C09098=1084.373,-43.335,-55.194,174.208,18.576,153.076
C09099=1084.367,-43.584,-55.182,174.206,18.574,153.076
C09100=1084.361,-43.833,-55.170,174.205,18.572,153.076
C09101=1084.355,-44.083,-55.158,174.204,18.571,153.076
C09102=1084.349,-44.333,-55.147,174.202,18.569,153.076
C09103=1084.343,-44.583,-55.134,174.201,18.568,153.076
C09104=1084.337,-44.833,-55.122,174.200,18.566,153.076
C09105=1084.331,-45.081,-55.110,174.198,18.565,153.076
C09106=1084.325,-45.331,-55.097,174.196,18.563,153.076
C09107=1084.320,-45.582,-55.086,174.195,18.561,153.076
C09108=1084.314,-45.831,-55.074,174.193,18.559,153.076
C09109=1084.308,-46.081,-55.061,174.192,18.557,153.076
C09110=1084.301,-46.330,-55.049,174.190,18.556,153.076
C09111=1084.296,-46.580,-55.038,174.189,18.554,153.076
C09112=1084.290,-46.830,-55.025,174.188,18.553,153.076
C09113=1084.284,-47.079,-55.014,174.186,18.551,153.076
C09114=1084.278,-47.329,-55.001,174.185,18.549,153.075
C09115=1084.272,-47.579,-54.990,174.183,18.547,153.075
C09116=1084.267,-47.828,-54.978,174.181,18.546,153.075
C09117=1084.260,-48.078,-54.966,174.180,18.544,153.075
C09118=1084.255,-48.327,-54.954,174.178,18.543,153.075
C09119=1084.249,-48.577,-54.942,174.177,18.541,153.075
C09120=1084.242,-48.850,-54.929,174.176,18.539,153.075
C09121=1084.236,-49.122,-54.916,174.174,18.537,153.075
C09122=1084.230,-49.395,-54.903,174.172,18.535,153.075
C09123=1084.223,-49.668,-54.890,174.171,18.534,153.075
C09124=1084.217,-49.917,-54.878,174.169,18.532,153.075
C09125=1084.211,-50.167,-54.866,174.168,18.531,153.075
C09126=1084.205,-50.416,-54.855,174.167,18.529,153.075
C09127=1084.199,-50.666,-54.842,174.164,18.527,153.075
C09128=1084.194,-50.915,-54.831,174.163,18.525,153.075
C09129=1084.187,-51.165,-54.819,174.162,18.524,153.075
C09130=1084.181,-51.415,-54.807,174.160,18.522,153.075
C09131=1084.175,-51.664,-54.796,174.158,18.521,153.075
C09132=1084.169,-51.914,-54.784,174.157,18.519,153.075
C09133=1084.163,-52.164,-54.771,174.156,18.518,153.075
C09134=1084.157,-52.413,-54.761,174.154,18.516,153.075
C09135=1084.150,-52.663,-54.749,174.153,18.515,153.075
C09136=1084.145,-52.913,-54.737,174.151,18.513,153.075
C09137=1084.139,-53.162,-54.725,174.150,18.512,153.075
C09138=1084.132,-53.412,-54.714,174.148,18.510,153.075
C09139=1084.127,-53.662,-54.702,174.147,18.509,153.075
C09140=1084.120,-53.911,-54.690,174.145,18.507,153.075
C09141=1084.114,-54.161,-54.679,174.143,18.505,153.075
C09142=1084.108,-54.410,-54.667,174.142,18.503,153.074
C09143=1084.102,-54.661,-54.655,174.140,18.502,153.074
C09144=1084.096,-54.910,-54.644,174.139,18.500,153.074
C09145=1084.090,-55.160,-54.632,174.138,18.499,153.074
C09146=1084.085,-55.409,-54.620,174.136,18.497,153.074
C09147=1084.078,-55.659,-54.609,174.135,18.496,153.074
C09148=1084.072,-55.909,-54.597,174.133,18.494,153.074
C09149=1084.066,-56.158,-54.586,174.132,18.493,153.074
C09150=1084.060,-56.408,-54.573,174.131,18.491,153.074
C09151=1084.054,-56.658,-54.563,174.129,18.490,153.074
C09152=1084.048,-56.907,-54.551,174.128,18.488,153.074
C09153=1084.042,-57.157,-54.540,174.126,18.486,153.074
C09154=1084.036,-57.407,-54.527,174.124,18.484,153.074
C09155=1084.030,-57.656,-54.516,174.123,18.483,153.074
C09156=1084.024,-57.906,-54.504,174.121,18.482,153.074
C09157=1084.018,-58.155,-54.493,174.119,18.480,153.074
C09158=1084.012,-58.405,-54.481,174.118,18.479,153.074
C09159=1084.006,-58.655,-54.470,174.117,18.477,153.074
C09160=1084.000,-58.905,-54.459,174.115,18.476,153.074
C09161=1083.993,-59.154,-54.447,174.114,18.474,153.074
C09162=1083.988,-59.404,-54.436,174.112,18.473,153.074
C09163=1083.982,-59.654,-54.423,174.111,18.471,153.074
C09164=1083.976,-59.903,-54.413,174.109,18.469,153.074
C09165=1083.970,-60.153,-54.401,174.108,18.468,153.074
C09166=1083.964,-60.402,-54.390,174.107,18.466,153.074
C09167=1083.958,-60.653,-54.378,174.105,18.465,153.074
C09168=1083.952,-60.902,-54.366,174.104,18.463,153.074
C09169=1083.946,-61.151,-54.355,174.102,18.462,153.074
C09170=1083.940,-61.401,-54.344,174.101,18.461,153.074
C09171=1083.934,-61.650,-54.333,174.099,18.459,153.074
C09172=1083.928,-61.901,-54.321,174.098,18.458,153.074
C09173=1083.922,-62.150,-54.310,174.096,18.456,153.074
C09174=1083.916,-62.400,-54.298,174.094,18.454,153.074
C09175=1083.910,-62.649,-54.287,174.093,18.452,153.074
C09176=1083.904,-62.899,-54.276,174.091,18.451,153.074
C09177=1083.899,-63.149,-54.264,174.090,18.449,153.074
C09178=1083.892,-63.399,-54.252,174.088,18.448,153.074
C09179=1083.886,-63.648,-54.241,174.087,18.447,153.074
C09180=1083.881,-63.898,-54.231,174.085,18.445,153.074
C09181=1083.874,-64.147,-54.219,174.084,18.444,153.074
C09182=1083.868,-64.397,-54.208,174.083,18.442,153.074
C09183=1083.863,-64.647,-54.196,174.081,18.441,153.074
C09184=1083.856,-64.921,-54.184,174.080,18.439,153.074
C09185=1083.850,-65.194,-54.171,174.078,18.438,153.074
C09186=1083.843,-65.469,-54.159,174.076,18.435,153.074
C09187=1083.837,-65.742,-54.147,174.075,18.434,153.073
C09188=1083.830,-65.993,-54.135,174.073,18.432,153.073
C09189=1083.824,-66.241,-54.124,174.071,18.431,153.074
C09190=1083.819,-66.491,-54.113,174.070,18.430,153.074
C09191=1083.812,-66.741,-54.102,174.069,18.428,153.073
C09192=1083.807,-66.991,-54.091,174.067,18.427,153.073
C09193=1083.800,-67.241,-54.080,174.066,18.425,153.073
C09194=1083.795,-67.490,-54.067,174.064,18.424,153.073
C09195=1083.789,-67.740,-54.056,174.063,18.422,153.073
C09196=1083.783,-67.990,-54.045,174.061,18.421,153.073
C09197=1083.777,-68.239,-54.034,174.060,18.420,153.073
C09198=1083.771,-68.489,-54.023,174.058,18.418,153.073
C09199=1083.765,-68.739,-54.012,174.057,18.416,153.073
C09200=1083.759,-68.988,-54.001,174.056,18.415,153.073
C09201=1083.753,-69.237,-53.990,174.054,18.413,153.073
C09202=1083.748,-69.488,-53.978,174.052,18.412,153.073
C09203=1083.742,-69.737,-53.967,174.051,18.411,153.073
C09204=1083.736,-69.987,-53.956,174.050,18.409,153.073
C09205=1083.730,-70.237,-53.945,174.048,18.408,153.073
C09206=1083.724,-70.486,-53.934,174.047,18.406,153.073
C09207=1083.718,-70.736,-53.923,174.045,18.405,153.073
C09208=1083.712,-70.986,-53.912,174.044,18.404,153.073
C09209=1083.706,-71.235,-53.900,174.042,18.402,153.073
C09210=1083.700,-71.484,-53.889,174.041,18.400,153.073
C09211=1083.694,-71.735,-53.878,174.039,18.399,153.073
C09212=1083.688,-71.984,-53.867,174.038,18.397,153.073
C09213=1083.683,-72.234,-53.856,174.036,18.396,153.073
C09214=1083.677,-72.483,-53.845,174.035,18.395,153.073
C09215=1083.671,-72.734,-53.834,174.033,18.393,153.073
C09216=1083.665,-72.983,-53.823,174.032,18.392,153.073
C09217=1083.660,-73.233,-53.812,174.031,18.390,153.073
C09218=1083.653,-73.483,-53.801,174.029,18.389,153.073
C09219=1083.647,-73.732,-53.790,174.028,18.388,153.073
C09220=1083.642,-73.982,-53.779,174.026,18.386,153.073
C09221=1083.636,-74.231,-53.768,174.025,18.384,153.073
C09222=1083.630,-74.481,-53.757,174.023,18.383,153.073
C09223=1083.624,-74.731,-53.746,174.022,18.382,153.073
C09224=1083.618,-74.980,-53.735,174.020,18.380,153.073
C09225=1083.611,-75.230,-53.724,174.018,18.379,153.073
C09226=1083.605,-75.480,-53.714,174.017,18.378,153.073
C09227=1083.600,-75.729,-53.703,174.016,18.376,153.073
C09228=1083.593,-75.979,-53.691,174.014,18.375,153.073
C09229=1083.588,-76.229,-53.681,174.013,18.374,153.073
C09230=1083.582,-76.478,-53.670,174.011,18.372,153.073
C09231=1083.575,-76.729,-53.658,174.009,18.371,153.073
C09232=1083.569,-76.978,-53.648,174.008,18.370,153.073
C09233=1083.563,-77.227,-53.637,174.007,18.368,153.073
C09234=1083.557,-77.477,-53.626,174.005,18.367,153.073
C09235=1083.551,-77.728,-53.616,174.003,18.365,153.073
C09236=1083.546,-77.977,-53.605,174.002,18.364,153.074
C09237=1083.540,-78.227,-53.594,174.000,18.363,153.074
C09238=1083.534,-78.476,-53.583,173.999,18.361,153.074
C09239=1083.527,-78.726,-53.573,173.997,18.360,153.074
C09240=1083.521,-78.975,-53.562,173.996,18.359,153.074
C09241=1083.516,-79.225,-53.551,173.994,18.357,153.074
C09242=1083.510,-79.474,-53.540,173.993,18.356,153.074
C09243=1083.504,-79.725,-53.529,173.991,18.355,153.074
C09244=1083.498,-79.975,-53.519,173.990,18.354,153.074
C09245=1083.492,-80.224,-53.508,173.988,18.352,153.074
C09246=1083.485,-80.474,-53.497,173.987,18.350,153.074
C09247=1083.480,-80.724,-53.486,173.985,18.349,153.074
C09248=1083.473,-81.000,-53.475,173.984,18.348,153.074
C09249=1083.466,-81.276,-53.463,173.982,18.347,153.074
C09250=1083.459,-81.552,-53.451,173.981,18.345,153.074
C09251=1083.452,-81.827,-53.440,173.979,18.344,153.074
C09252=1083.446,-82.078,-53.428,173.978,18.343,153.074
C09253=1083.440,-82.327,-53.418,173.976,18.342,153.074
C09254=1083.434,-82.577,-53.408,173.974,18.340,153.074
C09255=1083.428,-82.826,-53.397,173.973,18.339,153.074
C09256=1083.421,-83.076,-53.387,173.971,18.338,153.074
C09257=1083.416,-83.326,-53.376,173.970,18.337,153.074
C09258=1083.410,-83.575,-53.365,173.968,18.335,153.074
C09259=1083.404,-83.825,-53.355,173.967,18.334,153.074
C09260=1083.397,-84.075,-53.344,173.965,18.332,153.074
C09261=1083.392,-84.325,-53.333,173.963,18.331,153.074
C09262=1083.385,-84.574,-53.323,173.962,18.330,153.074
C09263=1083.380,-84.824,-53.313,173.960,18.329,153.074
C09264=1083.373,-85.074,-53.301,173.959,18.327,153.074
C09265=1083.367,-85.323,-53.291,173.957,18.326,153.075
C09266=1083.361,-85.573,-53.281,173.957,18.325,153.074
C09267=1083.355,-85.823,-53.271,173.955,18.324,153.075
C09268=1083.349,-86.073,-53.259,173.954,18.323,153.075
C09269=1083.343,-86.322,-53.249,173.952,18.322,153.075
C09270=1083.337,-86.572,-53.239,173.950,18.321,153.075
C09271=1083.331,-86.822,-53.228,173.949,18.319,153.075
C09272=1083.324,-87.071,-53.218,173.947,18.318,153.075
C09273=1083.318,-87.322,-53.207,173.946,18.316,153.075
C09274=1083.313,-87.571,-53.196,173.944,18.315,153.075
C09275=1083.306,-87.820,-53.186,173.943,18.314,153.075
C09276=1083.301,-88.070,-53.176,173.941,18.313,153.075
C09277=1083.294,-88.320,-53.166,173.939,18.312,153.075
C09278=1083.289,-88.569,-53.155,173.938,18.310,153.075
C09279=1083.282,-88.820,-53.145,173.936,18.309,153.075
C09280=1083.276,-89.069,-53.134,173.936,18.308,153.075
C09281=1083.271,-89.319,-53.124,173.934,18.307,153.075
C09282=1083.264,-89.568,-53.114,173.932,18.306,153.075
C09283=1083.258,-89.818,-53.103,173.931,18.305,153.075
C09284=1083.252,-90.068,-53.093,173.929,18.304,153.075
C09285=1083.246,-90.318,-53.082,173.928,18.302,153.075
C09286=1083.240,-90.568,-53.072,173.926,18.301,153.075
C09287=1083.234,-90.817,-53.061,173.925,18.299,153.075
C09288=1083.227,-91.066,-53.051,173.923,18.298,153.076
C09289=1083.222,-91.316,-53.041,173.921,18.297,153.076
C09290=1083.216,-91.566,-53.030,173.920,18.296,153.076
C09291=1083.210,-91.816,-53.021,173.919,18.295,153.076
C09292=1083.204,-92.065,-53.010,173.917,18.294,153.076
C09293=1083.198,-92.316,-53.000,173.916,18.293,153.076
C09294=1083.192,-92.565,-52.989,173.914,18.292,153.076
C09295=1083.186,-92.815,-52.979,173.913,18.290,153.076
C09296=1083.180,-93.064,-52.968,173.911,18.289,153.076
C09297=1083.174,-93.314,-52.959,173.909,18.288,153.076
C09298=1083.168,-93.564,-52.948,173.908,18.287,153.076
C09299=1083.162,-93.814,-52.938,173.906,18.286,153.076
C09300=1083.156,-94.063,-52.928,173.905,18.285,153.076
C09301=1083.150,-94.313,-52.918,173.904,18.284,153.076
C09302=1083.144,-94.562,-52.907,173.902,18.283,153.076
C09303=1083.138,-94.812,-52.897,173.901,18.281,153.076
C09304=1083.132,-95.062,-52.886,173.899,18.280,153.076
C09305=1083.126,-95.312,-52.877,173.898,18.279,153.077
C09306=1083.120,-95.562,-52.866,173.896,18.278,153.077
C09307=1083.114,-95.811,-52.856,173.895,18.276,153.077
C09308=1083.108,-96.061,-52.845,173.893,18.275,153.077
C09309=1083.102,-96.311,-52.836,173.891,18.274,153.077
C09310=1083.096,-96.561,-52.826,173.890,18.273,153.077
C09311=1083.090,-96.810,-52.815,173.889,18.272,153.077
C09312=1083.084,-97.089,-52.804,173.887,18.271,153.077
C09313=1083.077,-97.366,-52.793,173.885,18.270,153.077
C09314=1083.070,-97.645,-52.782,173.883,18.268,153.077
C09315=1083.063,-97.923,-52.770,173.882,18.267,153.077
C09316=1083.057,-98.173,-52.760,173.880,18.266,153.077
C09317=1083.051,-98.423,-52.749,173.878,18.265,153.077
C09318=1083.045,-98.672,-52.740,173.878,18.264,153.077
C09319=1083.039,-98.922,-52.730,173.876,18.263,153.077
C09320=1083.033,-99.172,-52.719,173.874,18.262,153.078
C09321=1083.027,-99.422,-52.710,173.873,18.261,153.078
C09322=1083.020,-99.672,-52.700,173.871,18.260,153.078
C09323=1083.014,-99.921,-52.690,173.870,18.258,153.078
C09324=1083.009,-100.171,-52.680,173.868,18.257,153.078
C09325=1083.002,-100.421,-52.670,173.867,18.257,153.078
C09326=1082.996,-100.670,-52.660,173.865,18.256,153.078
C09327=1082.990,-100.920,-52.650,173.864,18.255,153.078
C09328=1082.984,-101.170,-52.640,173.862,18.254,153.078
C09329=1082.978,-101.419,-52.630,173.860,18.253,153.078
C09330=1082.972,-101.669,-52.620,173.859,18.251,153.078
C09331=1082.966,-101.919,-52.610,173.857,18.250,153.079
C09332=1082.960,-102.168,-52.600,173.856,18.250,153.079
C09333=1082.954,-102.418,-52.590,173.855,18.249,153.079
C09334=1082.948,-102.668,-52.580,173.853,18.248,153.079
C09335=1082.942,-102.918,-52.570,173.851,18.247,153.079
C09336=1082.935,-103.167,-52.560,173.850,18.246,153.079
C09337=1082.929,-103.417,-52.551,173.848,18.244,153.079
C09338=1082.924,-103.667,-52.540,173.847,18.243,153.079
C09339=1082.918,-103.917,-52.531,173.846,18.242,153.079
C09340=1082.911,-104.166,-52.520,173.844,18.241,153.079
C09341=1082.905,-104.416,-52.511,173.842,18.240,153.079
C09342=1082.900,-104.666,-52.501,173.841,18.239,153.080
C09343=1082.893,-104.916,-52.491,173.839,18.238,153.080
C09344=1082.887,-105.165,-52.481,173.837,18.237,153.080
C09345=1082.881,-105.415,-52.471,173.837,18.237,153.080
C09346=1082.875,-105.665,-52.462,173.835,18.236,153.080
C09347=1082.869,-105.915,-52.452,173.833,18.235,153.080
C09348=1082.863,-106.165,-52.442,173.832,18.234,153.080
C09349=1082.857,-106.414,-52.432,173.830,18.232,153.080
C09350=1082.850,-106.664,-52.422,173.828,18.231,153.080
C09351=1082.844,-106.913,-52.413,173.828,18.231,153.080
C09352=1082.839,-107.164,-52.402,173.826,18.230,153.080
C09353=1082.833,-107.413,-52.393,173.824,18.229,153.081
C09354=1082.826,-107.663,-52.383,173.823,18.228,153.081
C09355=1082.820,-107.912,-52.373,173.821,18.227,153.081
C09356=1082.814,-108.162,-52.363,173.819,18.226,153.081
C09357=1082.808,-108.412,-52.354,173.818,18.225,153.081
C09358=1082.801,-108.662,-52.344,173.817,18.224,153.081
C09359=1082.795,-108.911,-52.335,173.815,18.223,153.081
C09360=1082.790,-109.162,-52.325,173.813,18.222,153.081
C09361=1082.784,-109.411,-52.315,173.812,18.221,153.081
C09362=1082.777,-109.661,-52.305,173.810,18.220,153.082
C09363=1082.771,-109.910,-52.295,173.809,18.220,153.082
C09364=1082.765,-110.160,-52.286,173.807,18.219,153.082
C09365=1082.759,-110.410,-52.276,173.806,18.218,153.082
C09366=1082.752,-110.660,-52.267,173.804,18.217,153.082
C09367=1082.746,-110.910,-52.257,173.802,18.216,153.082
C09368=1082.741,-111.159,-52.248,173.801,18.215,153.082
C09369=1082.735,-111.408,-52.238,173.800,18.214,153.082
C09370=1082.728,-111.658,-52.229,173.798,18.213,153.083
C09371=1082.722,-111.908,-52.219,173.796,18.212,153.083
C09372=1082.716,-112.158,-52.209,173.795,18.211,153.083
C09373=1082.710,-112.408,-52.200,173.794,18.211,153.083
C09374=1082.704,-112.658,-52.190,173.792,18.210,153.083
C09375=1082.698,-112.908,-52.180,173.790,18.209,153.083
C09376=1082.692,-113.181,-52.169,173.789,18.208,153.083
C09377=1082.684,-113.457,-52.159,173.787,18.207,153.083
C09378=1082.678,-113.731,-52.149,173.785,18.206,153.084
C09379=1082.671,-114.007,-52.138,173.783,18.205,153.084
C09380=1082.665,-114.256,-52.129,173.782,18.204,153.084
C09381=1082.659,-114.505,-52.119,173.781,18.203,153.084
C09382=1082.653,-114.755,-52.110,173.779,18.202,153.084
C09383=1082.647,-115.005,-52.100,173.778,18.201,153.084
C09384=1082.641,-115.255,-52.090,173.776,18.201,153.084
C09385=1082.635,-115.505,-52.081,173.774,18.200,153.084
C09386=1082.628,-115.754,-52.071,173.773,18.199,153.085
C09387=1082.622,-116.004,-52.062,173.771,18.198,153.085
C09388=1082.616,-116.254,-52.052,173.770,18.197,153.085
C09389=1082.609,-116.504,-52.043,173.768,18.196,153.085
C09390=1082.603,-116.753,-52.034,173.766,18.196,153.085
C09391=1082.597,-117.002,-52.024,173.765,18.195,153.085
C09392=1082.591,-117.252,-52.015,173.764,18.194,153.085
C09393=1082.585,-117.502,-52.005,173.762,18.193,153.085
C09394=1082.579,-117.752,-51.996,173.760,18.192,153.086
C09395=1082.573,-118.002,-51.987,173.759,18.192,153.086
C09396=1082.567,-118.252,-51.977,173.758,18.191,153.086
C09397=1082.561,-118.502,-51.968,173.756,18.190,153.086
C09398=1082.555,-118.752,-51.958,173.754,18.189,153.086
C09399=1082.549,-119.001,-51.949,173.753,18.189,153.086
C09400=1082.543,-119.251,-51.939,173.751,18.188,153.086
C09401=1082.536,-119.500,-51.930,173.750,18.187,153.087
C09402=1082.530,-119.750,-51.922,173.748,18.186,153.087
C09403=1082.524,-120.000,-51.912,173.746,18.186,153.087
C09404=1082.518,-120.250,-51.902,173.745,18.185,153.087
C09405=1082.512,-120.500,-51.893,173.744,18.184,153.087
C09406=1082.506,-120.749,-51.884,173.742,18.184,153.087
C09407=1082.500,-120.999,-51.874,173.740,18.183,153.088
C09408=1082.494,-121.248,-51.865,173.739,18.182,153.088
C09409=1082.487,-121.499,-51.856,173.737,18.181,153.088
C09410=1082.481,-121.748,-51.847,173.736,18.181,153.088
C09411=1082.475,-121.998,-51.837,173.734,18.180,153.088
C09412=1082.469,-122.247,-51.828,173.733,18.179,153.088
C09413=1082.463,-122.497,-51.818,173.731,18.179,153.088
C09414=1082.457,-122.748,-51.810,173.729,18.177,153.089
C09415=1082.450,-122.997,-51.801,173.728,18.176,153.089
C09416=1082.444,-123.247,-51.791,173.727,18.176,153.089
C09417=1082.438,-123.497,-51.781,173.725,18.175,153.089
C09418=1082.433,-123.746,-51.773,173.723,18.174,153.089
C09419=1082.426,-123.996,-51.763,173.721,18.174,153.089
C09420=1082.420,-124.246,-51.754,173.720,18.173,153.089
C09421=1082.413,-124.495,-51.745,173.719,18.172,153.090
C09422=1082.407,-124.746,-51.736,173.717,18.172,153.090
C09423=1082.402,-124.995,-51.727,173.716,18.171,153.090
C09424=1082.396,-125.245,-51.717,173.714,18.171,153.090
C09425=1082.389,-125.494,-51.708,173.712,18.170,153.090
C09426=1082.383,-125.745,-51.699,173.711,18.169,153.090
C09427=1082.377,-125.994,-51.690,173.710,18.169,153.091
C09428=1082.370,-126.243,-51.681,173.708,18.168,153.091
C09429=1082.364,-126.493,-51.672,173.706,18.167,153.091
C09430=1082.358,-126.743,-51.663,173.704,18.166,153.091
C09431=1082.352,-126.993,-51.653,173.703,18.166,153.091
C09432=1082.345,-127.243,-51.644,173.702,18.165,153.091
C09433=1082.340,-127.492,-51.636,173.700,18.164,153.092
C09434=1082.334,-127.742,-51.626,173.699,18.164,153.092
C09435=1082.327,-127.992,-51.617,173.697,18.163,153.092
C09436=1082.323,-128.248,-51.608,173.695,18.162,153.092
C09437=1082.323,-128.504,-51.596,173.695,18.160,153.092
C09438=1082.327,-128.758,-51.583,173.694,18.156,153.091
C09439=1082.334,-129.010,-51.570,173.694,18.152,153.090
C09440=1081.933,-129.032,-51.707,173.650,18.270,153.120
C09441=1081.926,-128.780,-51.721,173.650,18.275,153.121
C09442=1081.923,-128.525,-51.734,173.651,18.278,153.122
C09443=1081.922,-128.271,-51.745,173.652,18.280,153.122
C09444=1081.927,-128.014,-51.756,173.653,18.282,153.122
C09445=1081.932,-127.764,-51.764,173.655,18.283,153.122
C09446=1081.939,-127.515,-51.773,173.656,18.283,153.122
C09447=1081.945,-127.265,-51.783,173.658,18.284,153.122
C09448=1081.951,-127.015,-51.792,173.659,18.285,153.122
C09449=1081.957,-126.765,-51.801,173.661,18.285,153.121
C09450=1081.963,-126.516,-51.810,173.662,18.286,153.121
C09451=1081.969,-126.266,-51.819,173.664,18.286,153.121
C09452=1081.976,-126.016,-51.828,173.666,18.287,153.121
C09453=1081.982,-125.766,-51.837,173.667,18.287,153.121
C09454=1081.989,-125.517,-51.847,173.668,18.288,153.121
C09455=1081.994,-125.267,-51.855,173.670,18.289,153.120
C09456=1082.000,-125.017,-51.865,173.672,18.290,153.120
C09457=1082.007,-124.768,-51.874,173.673,18.290,153.120
C09458=1082.013,-124.517,-51.883,173.675,18.291,153.120
C09459=1082.019,-124.267,-51.892,173.676,18.292,153.120
C09460=1082.025,-124.018,-51.901,173.678,18.293,153.120
C09461=1082.031,-123.769,-51.910,173.679,18.293,153.120
C09462=1082.037,-123.518,-51.919,173.681,18.294,153.119
C09463=1082.044,-123.269,-51.929,173.683,18.295,153.119
C09464=1082.050,-123.019,-51.938,173.684,18.296,153.119
C09465=1082.056,-122.769,-51.948,173.685,18.296,153.119
C09466=1082.061,-122.520,-51.957,173.687,18.297,153.119
C09467=1082.068,-122.270,-51.965,173.689,18.298,153.119
C09468=1082.074,-122.020,-51.975,173.691,18.298,153.118
C09469=1082.080,-121.770,-51.984,173.692,18.299,153.118
C09470=1082.087,-121.520,-51.994,173.693,18.300,153.118
C09471=1082.093,-121.271,-52.004,173.695,18.301,153.118
C09472=1082.098,-121.021,-52.012,173.697,18.302,153.118
C09473=1082.104,-120.771,-52.022,173.698,18.302,153.118
C09474=1082.111,-120.522,-52.031,173.699,18.303,153.118
C09475=1082.117,-120.272,-52.040,173.701,18.304,153.117
C09476=1082.123,-120.022,-52.050,173.703,18.305,153.117
C09477=1082.130,-119.772,-52.059,173.705,18.306,153.117
C09478=1082.135,-119.523,-52.068,173.706,18.306,153.117
C09479=1082.141,-119.273,-52.077,173.707,18.307,153.117
C09480=1082.147,-119.023,-52.087,173.709,18.308,153.117
C09481=1082.153,-118.773,-52.096,173.711,18.309,153.117
C09482=1082.160,-118.524,-52.105,173.712,18.309,153.116
C09483=1082.166,-118.274,-52.115,173.713,18.310,153.116
C09484=1082.173,-118.024,-52.125,173.715,18.311,153.116
C09485=1082.179,-117.774,-52.134,173.717,18.312,153.116
C09486=1082.184,-117.525,-52.143,173.718,18.312,153.116
C09487=1082.191,-117.275,-52.153,173.719,18.313,153.116
C09488=1082.196,-117.025,-52.162,173.721,18.314,153.116
C09489=1082.203,-116.775,-52.171,173.723,18.315,153.116
C09490=1082.209,-116.525,-52.181,173.725,18.316,153.115
C09491=1082.215,-116.276,-52.190,173.726,18.316,153.115
C09492=1082.221,-116.026,-52.200,173.727,18.317,153.115
C09493=1082.227,-115.776,-52.210,173.729,18.318,153.115
C09494=1082.233,-115.526,-52.219,173.731,18.319,153.115
C09495=1082.239,-115.277,-52.228,173.732,18.320,153.115
C09496=1082.245,-115.027,-52.238,173.733,18.321,153.115
C09497=1082.251,-114.778,-52.248,173.735,18.321,153.114
C09498=1082.257,-114.528,-52.257,173.737,18.322,153.114
C09499=1082.264,-114.278,-52.267,173.738,18.323,153.114
C09500=1082.270,-114.028,-52.276,173.740,18.324,153.114
C09501=1082.277,-113.753,-52.287,173.742,18.325,153.114
C09502=1082.283,-113.478,-52.297,173.744,18.326,153.114
C09503=1082.290,-113.203,-52.308,173.744,18.327,153.114
C09504=1082.297,-112.928,-52.318,173.746,18.328,153.114
C09505=1082.303,-112.679,-52.327,173.748,18.329,153.114
C09506=1082.309,-112.429,-52.337,173.749,18.330,153.113
C09507=1082.315,-112.179,-52.346,173.751,18.331,153.113
C09508=1082.321,-111.929,-52.356,173.753,18.332,153.113
C09509=1082.328,-111.679,-52.366,173.754,18.333,153.113
C09510=1082.334,-111.430,-52.375,173.755,18.334,153.113
C09511=1082.340,-111.181,-52.385,173.757,18.334,153.113
C09512=1082.346,-110.930,-52.396,173.759,18.335,153.113
C09513=1082.352,-110.681,-52.405,173.761,18.336,153.113
C09514=1082.358,-110.431,-52.415,173.762,18.337,153.112
C09515=1082.364,-110.181,-52.424,173.763,18.338,153.112
C09516=1082.370,-109.931,-52.434,173.765,18.339,153.112
C09517=1082.377,-109.681,-52.443,173.766,18.340,153.112
C09518=1082.383,-109.432,-52.453,173.768,18.341,153.112
C09519=1082.389,-109.182,-52.463,173.770,18.342,153.112
C09520=1082.395,-108.932,-52.472,173.771,18.343,153.112
C09521=1082.402,-108.683,-52.482,173.772,18.343,153.112
C09522=1082.407,-108.434,-52.492,173.774,18.344,153.112
C09523=1082.413,-108.184,-52.501,173.776,18.345,153.111
C09524=1082.419,-107.934,-52.511,173.777,18.346,153.111
C09525=1082.425,-107.684,-52.521,173.779,18.347,153.111
C09526=1082.431,-107.434,-52.530,173.780,18.348,153.111
C09527=1082.437,-107.184,-52.540,173.782,18.349,153.111
C09528=1082.444,-106.935,-52.550,173.783,18.350,153.111
C09529=1082.450,-106.685,-52.560,173.785,18.351,153.111
C09530=1082.455,-106.435,-52.570,173.786,18.352,153.111
C09531=1082.461,-106.186,-52.580,173.788,18.353,153.111
C09532=1082.468,-105.936,-52.589,173.789,18.354,153.111
C09533=1082.474,-105.687,-52.599,173.791,18.355,153.111
C09534=1082.480,-105.437,-52.609,173.792,18.356,153.110
C09535=1082.486,-105.187,-52.619,173.794,18.357,153.110
C09536=1082.492,-104.937,-52.629,173.796,18.358,153.110
C09537=1082.498,-104.687,-52.638,173.797,18.359,153.110
C09538=1082.505,-104.438,-52.649,173.799,18.361,153.110
C09539=1082.510,-104.188,-52.659,173.800,18.361,153.110
C09540=1082.516,-103.938,-52.668,173.801,18.362,153.110
C09541=1082.522,-103.688,-52.678,173.803,18.363,153.110
C09542=1082.529,-103.439,-52.688,173.805,18.364,153.110
C09543=1082.534,-103.189,-52.698,173.806,18.365,153.110
C09544=1082.540,-102.939,-52.708,173.808,18.366,153.109
C09545=1082.547,-102.689,-52.717,173.809,18.368,153.110
C09546=1082.553,-102.440,-52.728,173.810,18.368,153.109
C09547=1082.559,-102.190,-52.738,173.812,18.369,153.109
C09548=1082.565,-101.940,-52.747,173.814,18.370,153.109
C09549=1082.571,-101.691,-52.758,173.815,18.371,153.109
C09550=1082.577,-101.441,-52.767,173.817,18.372,153.109
C09551=1082.583,-101.191,-52.777,173.818,18.374,153.109
C09552=1082.590,-100.941,-52.788,173.820,18.375,153.109
C09553=1082.596,-100.691,-52.798,173.821,18.375,153.109
C09554=1082.601,-100.441,-52.808,173.823,18.376,153.109
C09555=1082.608,-100.192,-52.818,173.824,18.377,153.109
C09556=1082.614,-99.942,-52.828,173.826,18.379,153.109
C09557=1082.620,-99.692,-52.838,173.827,18.380,153.109
C09558=1082.626,-99.443,-52.848,173.829,18.381,153.108
C09559=1082.632,-99.193,-52.858,173.831,18.382,153.108
C09560=1082.638,-98.944,-52.867,173.832,18.382,153.108
C09561=1082.644,-98.694,-52.878,173.833,18.384,153.108
C09562=1082.650,-98.444,-52.888,173.835,18.385,153.108
C09563=1082.656,-98.194,-52.897,173.836,18.386,153.108
C09564=1082.662,-97.945,-52.908,173.838,18.387,153.108
C09565=1082.670,-97.666,-52.919,173.839,18.389,153.108
C09566=1082.676,-97.388,-52.931,173.841,18.390,153.108
C09567=1082.683,-97.109,-52.942,173.843,18.391,153.108
C09568=1082.689,-96.830,-52.953,173.844,18.392,153.108
C09569=1082.695,-96.581,-52.964,173.846,18.393,153.108
C09570=1082.702,-96.331,-52.973,173.848,18.394,153.108
C09571=1082.707,-96.082,-52.984,173.849,18.396,153.108
C09572=1082.714,-95.832,-52.994,173.851,18.397,153.107
C09573=1082.719,-95.582,-53.004,173.852,18.398,153.107
C09574=1082.725,-95.333,-53.014,173.854,18.399,153.107
C09575=1082.731,-95.083,-53.025,173.855,18.400,153.107
C09576=1082.737,-94.833,-53.034,173.857,18.402,153.107
C09577=1082.743,-94.583,-53.045,173.858,18.402,153.107
C09578=1082.749,-94.334,-53.055,173.859,18.403,153.107
C09579=1082.755,-94.083,-53.065,173.861,18.405,153.107
C09580=1082.761,-93.834,-53.076,173.863,18.406,153.107
C09581=1082.767,-93.584,-53.086,173.864,18.407,153.107
C09582=1082.773,-93.334,-53.097,173.866,18.409,153.107
C09583=1082.779,-93.085,-53.106,173.867,18.410,153.107
C09584=1082.785,-92.835,-53.117,173.869,18.411,153.107
C09585=1082.791,-92.586,-53.127,173.870,18.412,153.107
C09586=1082.797,-92.336,-53.138,173.872,18.413,153.107
C09587=1082.803,-92.087,-53.148,173.874,18.415,153.107
C09588=1082.809,-91.837,-53.158,173.874,18.415,153.107
C09589=1082.816,-91.587,-53.169,173.876,18.417,153.107
C09590=1082.821,-91.337,-53.179,173.877,18.418,153.106
C09591=1082.828,-91.087,-53.189,173.879,18.419,153.106
C09592=1082.833,-90.837,-53.199,173.881,18.420,153.106
C09593=1082.840,-90.588,-53.210,173.882,18.421,153.106
C09594=1082.845,-90.339,-53.220,173.884,18.423,153.106
C09595=1082.851,-90.089,-53.231,173.885,18.424,153.106
C09596=1082.858,-89.839,-53.241,173.887,18.426,153.106
C09597=1082.863,-89.589,-53.251,173.888,18.427,153.106
C09598=1082.870,-89.339,-53.262,173.890,18.428,153.106
C09599=1082.875,-89.090,-53.273,173.892,18.429,153.106
C09600=1082.882,-88.840,-53.282,173.892,18.430,153.106
C09601=1082.887,-88.591,-53.293,173.894,18.431,153.106
C09602=1082.893,-88.340,-53.304,173.896,18.432,153.106
C09603=1082.900,-88.091,-53.314,173.897,18.434,153.106
C09604=1082.906,-87.841,-53.325,173.899,18.435,153.106
C09605=1082.912,-87.591,-53.334,173.900,18.436,153.106
C09606=1082.918,-87.342,-53.345,173.902,18.437,153.106
C09607=1082.923,-87.092,-53.356,173.903,18.439,153.106
C09608=1082.930,-86.842,-53.366,173.905,18.440,153.106
C09609=1082.936,-86.592,-53.377,173.906,18.441,153.106
C09610=1082.942,-86.343,-53.387,173.908,18.442,153.106
C09611=1082.948,-86.094,-53.398,173.909,18.444,153.106
C09612=1082.954,-85.843,-53.409,173.911,18.445,153.105
C09613=1082.961,-85.594,-53.419,173.912,18.447,153.106
C09614=1082.966,-85.344,-53.430,173.913,18.447,153.105
C09615=1082.972,-85.094,-53.439,173.915,18.449,153.106
C09616=1082.978,-84.845,-53.450,173.916,18.450,153.105
C09617=1082.985,-84.595,-53.461,173.918,18.451,153.105
C09618=1082.991,-84.346,-53.472,173.920,18.452,153.105
C09619=1082.996,-84.095,-53.482,173.921,18.454,153.105
C09620=1083.003,-83.846,-53.492,173.923,18.455,153.105
C09621=1083.009,-83.596,-53.503,173.924,18.456,153.105
C09622=1083.015,-83.347,-53.514,173.926,18.457,153.105
C09623=1083.021,-83.097,-53.524,173.927,18.459,153.105
C09624=1083.027,-82.847,-53.535,173.929,18.460,153.105
C09625=1083.033,-82.597,-53.546,173.930,18.461,153.105
C09626=1083.040,-82.348,-53.556,173.932,18.462,153.105
C09627=1083.045,-82.098,-53.567,173.933,18.464,153.105
C09628=1083.051,-81.848,-53.578,173.935,18.465,153.105
C09629=1083.058,-81.573,-53.590,173.937,18.467,153.105
C09630=1083.065,-81.296,-53.601,173.938,18.468,153.105
C09631=1083.072,-81.020,-53.613,173.940,18.469,153.105
C09632=1083.078,-80.743,-53.625,173.941,18.471,153.105
C09633=1083.085,-80.494,-53.635,173.943,18.472,153.105
C09634=1083.091,-80.244,-53.646,173.944,18.473,153.105
C09635=1083.097,-79.995,-53.657,173.946,18.475,153.105
C09636=1083.104,-79.745,-53.668,173.947,18.476,153.105
C09637=1083.109,-79.495,-53.678,173.949,18.477,153.105
C09638=1083.115,-79.245,-53.689,173.950,18.479,153.105
C09639=1083.121,-78.996,-53.700,173.952,18.480,153.105
C09640=1083.127,-78.745,-53.711,173.953,18.481,153.105
C09641=1083.133,-78.496,-53.722,173.955,18.483,153.105
C09642=1083.139,-78.247,-53.732,173.956,18.484,153.105
C09643=1083.145,-77.997,-53.743,173.958,18.485,153.105
C09644=1083.151,-77.747,-53.754,173.959,18.487,153.105
C09645=1083.157,-77.498,-53.765,173.961,18.488,153.105
C09646=1083.163,-77.248,-53.776,173.962,18.490,153.105
C09647=1083.169,-76.997,-53.786,173.964,18.491,153.105
C09648=1083.175,-76.748,-53.797,173.965,18.492,153.105
C09649=1083.181,-76.499,-53.808,173.967,18.494,153.105
C09650=1083.187,-76.249,-53.819,173.968,18.495,153.105
C09651=1083.193,-75.999,-53.830,173.970,18.496,153.104
C09652=1083.199,-75.749,-53.841,173.971,18.498,153.105
C09653=1083.204,-75.500,-53.852,173.973,18.499,153.105
C09654=1083.211,-75.250,-53.863,173.974,18.501,153.105
C09655=1083.217,-75.000,-53.874,173.976,18.502,153.104
C09656=1083.223,-74.751,-53.884,173.977,18.503,153.105
C09657=1083.229,-74.501,-53.895,173.979,18.505,153.105
C09658=1083.235,-74.251,-53.906,173.980,18.506,153.104
C09659=1083.241,-74.002,-53.917,173.982,18.508,153.104
C09660=1083.247,-73.752,-53.928,173.983,18.509,153.104
C09661=1083.253,-73.502,-53.939,173.985,18.511,153.105
C09662=1083.259,-73.253,-53.950,173.986,18.512,153.105
C09663=1083.264,-73.003,-53.961,173.988,18.513,153.104
C09664=1083.271,-72.753,-53.972,173.989,18.515,153.104
C09665=1083.276,-72.504,-53.983,173.991,18.516,153.105
C09666=1083.281,-72.254,-53.994,173.992,18.518,153.105
C09667=1083.288,-72.004,-54.006,173.994,18.519,153.105
C09668=1083.294,-71.755,-54.017,173.995,18.521,153.105
C09669=1083.300,-71.505,-54.028,173.997,18.522,153.105
C09670=1083.305,-71.256,-54.039,173.998,18.523,153.105
C09671=1083.312,-71.006,-54.050,174.000,18.525,153.105
C09672=1083.317,-70.756,-54.061,174.001,18.527,153.105
C09673=1083.323,-70.507,-54.072,174.002,18.528,153.105
C09674=1083.330,-70.256,-54.083,174.004,18.530,153.105
C09675=1083.335,-70.007,-54.094,174.005,18.531,153.105
C09676=1083.341,-69.757,-54.105,174.007,18.533,153.105
C09677=1083.347,-69.507,-54.117,174.008,18.534,153.105
C09678=1083.353,-69.258,-54.128,174.010,18.535,153.105
C09679=1083.358,-69.009,-54.139,174.011,18.537,153.105
C09680=1083.365,-68.758,-54.151,174.013,18.538,153.105
C09681=1083.370,-68.509,-54.161,174.014,18.540,153.105
C09682=1083.376,-68.259,-54.172,174.015,18.541,153.105
C09683=1083.383,-68.009,-54.184,174.017,18.543,153.105
C09684=1083.388,-67.760,-54.194,174.018,18.545,153.105
C09685=1083.394,-67.511,-54.207,174.020,18.546,153.105
C09686=1083.400,-67.260,-54.218,174.021,18.547,153.105
C09687=1083.406,-67.011,-54.229,174.023,18.549,153.105
C09688=1083.412,-66.761,-54.240,174.024,18.550,153.105
C09689=1083.418,-66.511,-54.251,174.026,18.552,153.105
C09690=1083.424,-66.262,-54.262,174.027,18.553,153.105
C09691=1083.430,-66.012,-54.274,174.029,18.555,153.105
C09692=1083.436,-65.763,-54.285,174.030,18.556,153.105
C09693=1083.442,-65.488,-54.298,174.032,18.558,153.105
C09694=1083.448,-65.214,-54.310,174.034,18.560,153.105
C09695=1083.455,-64.940,-54.323,174.035,18.561,153.105
C09696=1083.462,-64.666,-54.335,174.037,18.563,153.105
C09697=1083.468,-64.416,-54.346,174.038,18.565,153.105
C09698=1083.474,-64.167,-54.357,174.039,18.566,153.105
C09699=1083.480,-63.918,-54.368,174.041,18.568,153.105
C09700=1083.486,-63.668,-54.380,174.043,18.569,153.105
C09701=1083.491,-63.418,-54.391,174.045,18.571,153.105
C09702=1083.498,-63.168,-54.403,174.046,18.572,153.105
C09703=1083.503,-62.919,-54.414,174.048,18.574,153.105
C09704=1083.510,-62.669,-54.425,174.049,18.575,153.105
C09705=1083.515,-62.419,-54.436,174.051,18.577,153.105
C09706=1083.521,-62.169,-54.449,174.052,18.578,153.105
C09707=1083.527,-61.920,-54.460,174.053,18.580,153.105
C09708=1083.533,-61.670,-54.470,174.055,18.581,153.105
C09709=1083.540,-61.421,-54.482,174.056,18.583,153.105
C09710=1083.545,-61.171,-54.493,174.058,18.585,153.105
C09711=1083.551,-60.921,-54.506,174.059,18.586,153.105
C09712=1083.557,-60.672,-54.517,174.061,18.588,153.105
C09713=1083.563,-60.422,-54.528,174.062,18.589,153.105
C09714=1083.569,-60.173,-54.540,174.063,18.591,153.105
C09715=1083.576,-59.923,-54.551,174.065,18.592,153.106
C09716=1083.581,-59.673,-54.562,174.066,18.594,153.106
C09717=1083.587,-59.423,-54.574,174.068,18.595,153.106
C09718=1083.593,-59.174,-54.585,174.069,18.597,153.106
C09719=1083.600,-58.924,-54.597,174.071,18.598,153.106
C09720=1083.605,-58.674,-54.609,174.073,18.600,153.106
C09721=1083.611,-58.425,-54.620,174.074,18.601,153.106
C09722=1083.617,-58.175,-54.631,174.076,18.603,153.106
C09723=1083.623,-57.925,-54.643,174.077,18.605,153.106
C09724=1083.629,-57.676,-54.655,174.079,18.606,153.106
C09725=1083.635,-57.426,-54.666,174.080,18.608,153.106
C09726=1083.642,-57.176,-54.678,174.082,18.609,153.106
C09727=1083.647,-56.927,-54.689,174.083,18.611,153.106
C09728=1083.653,-56.677,-54.701,174.084,18.612,153.106
C09729=1083.659,-56.427,-54.712,174.086,18.614,153.106
C09730=1083.666,-56.178,-54.724,174.087,18.615,153.106
C09731=1083.671,-55.928,-54.735,174.089,18.617,153.106
C09732=1083.677,-55.678,-54.748,174.090,18.618,153.106
C09733=1083.683,-55.429,-54.759,174.092,18.620,153.106
C09734=1083.690,-55.179,-54.771,174.093,18.621,153.106
C09735=1083.696,-54.929,-54.782,174.095,18.624,153.106
C09736=1083.701,-54.680,-54.794,174.097,18.625,153.106
C09737=1083.708,-54.430,-54.805,174.098,18.627,153.106
C09738=1083.714,-54.181,-54.817,174.100,18.628,153.106
C09739=1083.720,-53.931,-54.829,174.101,18.630,153.106
C09740=1083.726,-53.681,-54.841,174.102,18.631,153.106
C09741=1083.732,-53.432,-54.852,174.104,18.633,153.106
C09742=1083.738,-53.182,-54.863,174.105,18.634,153.106
C09743=1083.744,-52.933,-54.876,174.107,18.636,153.106
C09744=1083.750,-52.682,-54.887,174.108,18.637,153.106
C09745=1083.757,-52.433,-54.899,174.109,18.639,153.106
C09746=1083.762,-52.184,-54.911,174.111,18.641,153.107
C09747=1083.768,-51.933,-54.922,174.112,18.643,153.107
C09748=1083.775,-51.684,-54.934,174.115,18.645,153.107
C09749=1083.780,-51.435,-54.946,174.116,18.646,153.107
C09750=1083.787,-51.184,-54.958,174.117,18.648,153.107
C09751=1083.793,-50.936,-54.969,174.119,18.649,153.107
C09752=1083.798,-50.685,-54.981,174.120,18.651,153.107
C09753=1083.805,-50.436,-54.993,174.122,18.652,153.107
C09754=1083.811,-50.187,-55.005,174.123,18.654,153.107
C09755=1083.817,-49.936,-55.016,174.125,18.655,153.107
C09756=1083.822,-49.687,-55.029,174.126,18.657,153.107
C09757=1083.829,-49.414,-55.042,174.128,18.659,153.107
C09758=1083.835,-49.141,-55.055,174.129,18.661,153.107
C09759=1083.842,-48.869,-55.068,174.131,18.663,153.107
C09760=1083.848,-48.596,-55.081,174.132,18.664,153.107
C09761=1083.854,-48.346,-55.093,174.134,18.667,153.107
C09762=1083.860,-48.096,-55.105,174.136,18.668,153.107
C09763=1083.866,-47.847,-55.117,174.137,18.670,153.107
C09764=1083.872,-47.598,-55.129,174.139,18.671,153.107
C09765=1083.877,-47.348,-55.140,174.140,18.673,153.107
C09766=1083.884,-47.098,-55.152,174.141,18.674,153.107
C09767=1083.890,-46.848,-55.165,174.143,18.676,153.108
C09768=1083.895,-46.599,-55.177,174.144,18.678,153.108
C09769=1083.901,-46.349,-55.188,174.146,18.679,153.108
C09770=1083.907,-46.100,-55.200,174.148,18.681,153.108
C09771=1083.913,-45.850,-55.212,174.149,18.683,153.108
C09772=1083.919,-45.600,-55.225,174.150,18.685,153.108
C09773=1083.924,-45.351,-55.236,174.152,18.687,153.108
C09774=1083.931,-45.101,-55.248,174.153,18.688,153.108
C09775=1083.937,-44.851,-55.261,174.155,18.690,153.108
C09776=1083.943,-44.602,-55.272,174.156,18.691,153.108
C09777=1083.949,-44.352,-55.285,174.157,18.693,153.108
C09778=1083.954,-44.102,-55.297,174.159,18.695,153.108
C09779=1083.960,-43.853,-55.308,174.161,18.697,153.108
C09780=1083.966,-43.603,-55.321,174.162,18.698,153.108
C09781=1083.972,-43.353,-55.333,174.164,18.700,153.108
C09782=1083.978,-43.104,-55.345,174.165,18.702,153.108
C09783=1083.984,-42.854,-55.358,174.167,18.704,153.108
C09784=1083.990,-42.605,-55.370,174.168,18.705,153.108
C09785=1083.996,-42.355,-55.381,174.169,18.707,153.109
C09786=1084.002,-42.105,-55.394,174.171,18.709,153.109
C09787=1084.008,-41.856,-55.406,174.173,18.711,153.109
C09788=1084.014,-41.606,-55.418,174.174,18.712,153.109
C09789=1084.020,-41.357,-55.430,174.176,18.714,153.109
C09790=1084.026,-41.107,-55.442,174.177,18.715,153.109
C09791=1084.032,-40.857,-55.455,174.178,18.717,153.109
C09792=1084.038,-40.608,-55.467,174.180,18.719,153.109
C09793=1084.044,-40.358,-55.479,174.181,18.720,153.109
C09794=1084.050,-40.108,-55.492,174.183,18.722,153.109
C09795=1084.056,-39.859,-55.504,174.185,18.724,153.109
C09796=1084.062,-39.610,-55.516,174.186,18.726,153.109
C09797=1084.068,-39.359,-55.528,174.188,18.728,153.109
C09798=1084.074,-39.109,-55.540,174.189,18.729,153.109
C09799=1084.080,-38.860,-55.552,174.190,18.731,153.109
C09800=1084.085,-38.611,-55.564,174.192,18.733,153.110
C09801=1084.091,-38.361,-55.577,174.193,18.734,153.110
C09802=1084.097,-38.111,-55.589,174.195,18.736,153.110
C09803=1084.103,-37.862,-55.602,174.196,18.738,153.110
C09804=1084.109,-37.612,-55.614,174.198,18.740,153.110
C09805=1084.115,-37.362,-55.626,174.199,18.741,153.110
C09806=1084.121,-37.112,-55.639,174.201,18.743,153.110
C09807=1084.126,-36.863,-55.651,174.202,18.745,153.110
C09808=1084.132,-36.613,-55.663,174.203,18.747,153.110
C09809=1084.138,-36.363,-55.676,174.205,18.749,153.110
C09810=1084.144,-36.115,-55.689,174.207,18.751,153.110
C09811=1084.150,-35.865,-55.701,174.208,18.752,153.110
C09812=1084.156,-35.615,-55.713,174.210,18.754,153.110
C09813=1084.162,-35.365,-55.726,174.211,18.756,153.111
C09814=1084.168,-35.116,-55.738,174.212,18.757,153.111
C09815=1084.173,-34.866,-55.751,174.214,18.759,153.111
C09816=1084.179,-34.616,-55.763,174.216,18.761,153.111
C09817=1084.185,-34.367,-55.776,174.217,18.763,153.111
C09818=1084.191,-34.117,-55.788,174.219,18.764,153.111
C09819=1084.197,-33.867,-55.800,174.220,18.767,153.111
C09820=1084.203,-33.618,-55.812,174.221,18.768,153.111
C09821=1084.209,-33.345,-55.827,174.223,18.771,153.111
C09822=1084.216,-33.074,-55.840,174.225,18.772,153.111
C09823=1084.222,-32.801,-55.854,174.226,18.774,153.111
C09824=1084.229,-32.529,-55.868,174.228,18.776,153.111
C09825=1084.235,-32.279,-55.880,174.230,18.778,153.111
C09826=1084.240,-32.030,-55.893,174.231,18.780,153.112
C09827=1084.246,-31.780,-55.905,174.232,18.781,153.112
C09828=1084.252,-31.530,-55.918,174.234,18.783,153.112
C09829=1084.258,-31.280,-55.931,174.235,18.785,153.112
C09830=1084.265,-31.031,-55.943,174.237,18.787,153.112
C09831=1084.271,-30.781,-55.955,174.239,18.789,153.112
C09832=1084.276,-30.532,-55.968,174.240,18.791,153.112
C09833=1084.282,-30.282,-55.980,174.241,18.792,153.112
C09834=1084.288,-30.033,-55.993,174.243,18.794,153.112
C09835=1084.294,-29.783,-56.006,174.244,18.796,153.112
C09836=1084.300,-29.533,-56.019,174.246,18.798,153.112
C09837=1084.306,-29.283,-56.031,174.248,18.799,153.112
C09838=1084.311,-29.034,-56.044,174.249,18.801,153.112
C09839=1084.317,-28.785,-56.057,174.250,18.803,153.113
C09840=1084.323,-28.535,-56.069,174.252,18.804,153.113
C09841=1084.329,-28.285,-56.082,174.253,18.806,153.113
C09842=1084.335,-28.036,-56.095,174.255,18.808,153.113
C09843=1084.341,-27.786,-56.108,174.257,18.810,153.113
C09844=1084.347,-27.536,-56.120,174.258,18.812,153.113
C09845=1084.353,-27.287,-56.133,174.259,18.814,153.113
C09846=1084.359,-27.037,-56.146,174.261,18.815,153.113
C09847=1084.365,-26.787,-56.158,174.263,18.818,153.113
C09848=1084.371,-26.538,-56.171,174.264,18.819,153.113
C09849=1084.377,-26.288,-56.184,174.265,18.821,153.113
C09850=1084.383,-26.038,-56.196,174.267,18.823,153.113
C09851=1084.389,-25.789,-56.210,174.268,18.825,153.114
C09852=1084.395,-25.539,-56.222,174.269,18.826,153.114
C09853=1084.400,-25.290,-56.234,174.272,18.828,153.114
C09854=1084.405,-25.041,-56.248,174.273,18.830,153.114
C09855=1084.411,-24.791,-56.261,174.274,18.832,153.114
C09856=1084.417,-24.541,-56.273,174.275,18.834,153.114
C09857=1084.423,-24.292,-56.287,174.277,18.836,153.114
C09858=1084.429,-24.042,-56.299,174.279,18.838,153.114
C09859=1084.436,-23.792,-56.313,174.280,18.840,153.114
C09860=1084.441,-23.542,-56.326,174.281,18.842,153.114
C09861=1084.446,-23.293,-56.338,174.283,18.843,153.114
C09862=1084.452,-23.044,-56.351,174.284,18.845,153.115
C09863=1084.458,-22.794,-56.364,174.286,18.847,153.115
C09864=1084.464,-22.545,-56.377,174.288,18.849,153.115
C09865=1084.470,-22.295,-56.390,174.289,18.851,153.115
C09866=1084.476,-22.045,-56.403,174.290,18.852,153.115
C09867=1084.482,-21.795,-56.416,174.292,18.855,153.115
C09868=1084.488,-21.545,-56.429,174.294,18.857,153.115
C09869=1084.494,-21.296,-56.442,174.295,18.858,153.115
C09870=1084.500,-21.046,-56.454,174.297,18.860,153.115
C09871=1084.505,-20.797,-56.468,174.298,18.862,153.115
C09872=1084.511,-20.547,-56.480,174.299,18.864,153.116
C09873=1084.517,-20.298,-56.494,174.301,18.865,153.116
C09874=1084.523,-20.048,-56.506,174.303,18.868,153.116
C09875=1084.529,-19.799,-56.519,174.304,18.869,153.116
C09876=1084.534,-19.549,-56.533,174.305,18.871,153.116
C09877=1084.540,-19.300,-56.546,174.307,18.873,153.116
C09878=1084.546,-19.050,-56.558,174.309,18.875,153.116
C09879=1084.552,-18.800,-56.572,174.310,18.877,153.116
C09880=1084.559,-18.551,-56.585,174.312,18.879,153.116
C09881=1084.564,-18.301,-56.598,174.313,18.881,153.116
C09882=1084.570,-18.052,-56.611,174.314,18.882,153.116
C09883=1084.576,-17.802,-56.624,174.316,18.885,153.117
C09884=1084.582,-17.553,-56.637,174.318,18.886,153.117
C09885=1084.589,-17.279,-56.652,174.319,18.888,153.117
C09886=1084.595,-17.007,-56.666,174.321,18.890,153.117
C09887=1084.602,-16.733,-56.680,174.322,18.892,153.117
C09888=1084.608,-16.460,-56.694,174.324,18.894,153.117
C09889=1084.613,-16.210,-56.708,174.326,18.896,153.117
C09890=1084.619,-15.961,-56.721,174.327,18.898,153.117
C09891=1084.625,-15.711,-56.734,174.329,18.900,153.117
C09892=1084.631,-15.461,-56.748,174.330,18.902,153.117
C09893=1084.638,-15.212,-56.761,174.331,18.904,153.118
C09894=1084.644,-14.962,-56.774,174.333,18.906,153.118
C09895=1084.649,-14.712,-56.788,174.335,18.908,153.118
C09896=1084.655,-14.462,-56.800,174.336,18.909,153.118
C09897=1084.661,-14.214,-56.813,174.337,18.911,153.118
C09898=1084.666,-13.964,-56.827,174.340,18.913,153.118
C09899=1084.672,-13.715,-56.840,174.341,18.915,153.118
C09900=1084.677,-13.465,-56.854,174.342,18.917,153.118
C09901=1084.684,-13.215,-56.867,174.343,18.919,153.118
C09902=1084.689,-12.966,-56.881,174.345,18.920,153.118
C09903=1084.695,-12.716,-56.893,174.347,18.923,153.119
C09904=1084.701,-12.467,-56.907,174.348,18.925,153.119
C09905=1084.707,-12.216,-56.921,174.349,18.927,153.119
C09906=1084.713,-11.967,-56.934,174.351,18.928,153.119
C09907=1084.719,-11.717,-56.947,174.353,18.931,153.119
C09908=1084.725,-11.468,-56.960,174.354,18.932,153.119
C09909=1084.730,-11.218,-56.974,174.356,18.934,153.119
C09910=1084.737,-10.969,-56.988,174.357,18.936,153.119
C09911=1084.742,-10.719,-57.001,174.358,18.938,153.119
C09912=1084.748,-10.469,-57.014,174.360,18.940,153.119
C09913=1084.753,-10.220,-57.028,174.362,18.942,153.120
C09914=1084.760,-9.971,-57.041,174.363,18.943,153.120
C09915=1084.765,-9.721,-57.055,174.364,18.945,153.120
C09916=1084.771,-9.471,-57.068,174.367,18.947,153.120
C09917=1084.777,-9.222,-57.081,174.368,18.950,153.120
C09918=1084.783,-8.972,-57.095,174.369,18.951,153.120
C09919=1084.789,-8.723,-57.108,174.370,18.953,153.120
C09920=1084.794,-8.473,-57.122,174.373,18.955,153.120
C09921=1084.801,-8.224,-57.135,174.374,18.957,153.120
C09922=1084.806,-7.974,-57.148,174.375,18.959,153.121
C09923=1084.813,-7.724,-57.162,174.377,18.961,153.121
C09924=1084.818,-7.474,-57.176,174.379,18.963,153.121
C09925=1084.824,-7.225,-57.189,174.380,18.965,153.121
C09926=1084.830,-6.976,-57.203,174.381,18.967,153.121
C09927=1084.836,-6.726,-57.216,174.383,18.968,153.121
C09928=1084.841,-6.477,-57.230,174.384,18.970,153.121
C09929=1084.847,-6.227,-57.244,174.386,18.972,153.121
C09930=1084.853,-5.978,-57.257,174.387,18.975,153.121
C09931=1084.859,-5.728,-57.271,174.389,18.976,153.121
C09932=1084.865,-5.478,-57.285,174.390,18.978,153.122
C09933=1084.871,-5.228,-57.298,174.392,18.980,153.122
C09934=1084.877,-4.979,-57.311,174.393,18.982,153.122
C09935=1084.882,-4.729,-57.325,174.395,18.984,153.122
C09936=1084.888,-4.480,-57.338,174.396,18.986,153.122
C09937=1084.894,-4.230,-57.352,174.398,18.988,153.122
C09938=1084.901,-3.980,-57.366,174.400,18.990,153.122
C09939=1084.906,-3.731,-57.380,174.401,18.991,153.122
C09940=1084.912,-3.482,-57.393,174.402,18.993,153.122
C09941=1084.918,-3.232,-57.407,174.405,18.995,153.122
C09942=1084.923,-2.982,-57.421,174.406,18.997,153.123
C09943=1084.929,-2.733,-57.434,174.407,18.999,153.123
C09944=1084.935,-2.484,-57.448,174.408,19.001,153.123
C09945=1084.941,-2.233,-57.462,174.411,19.003,153.123
C09946=1084.947,-1.984,-57.476,174.412,19.005,153.123
C09947=1084.952,-1.734,-57.490,174.413,19.007,153.123
C09948=1084.959,-1.486,-57.504,174.414,19.009,153.123
C09949=1084.964,-1.210,-57.519,174.417,19.011,153.123
C09950=1084.971,-0.935,-57.534,174.418,19.013,153.123
C09951=1084.977,-0.661,-57.550,174.420,19.016,153.124
C09952=1084.984,-0.386,-57.564,174.421,19.017,153.124
C09953=1084.989,-0.136,-57.578,174.423,19.020,153.124
C09954=1084.995,0.113,-57.592,174.425,19.021,153.124
C09955=1085.001,0.363,-57.605,174.426,19.023,153.124
C09956=1085.007,0.612,-57.620,174.427,19.025,153.124
C09957=1085.013,0.862,-57.634,174.429,19.028,153.124
C09958=1085.018,1.111,-57.648,174.431,19.030,153.124
C09959=1085.024,1.361,-57.662,174.432,19.031,153.124
C09960=1085.030,1.610,-57.675,174.434,19.034,153.125
C09961=1085.035,1.860,-57.689,174.435,19.036,153.125
C09962=1085.041,2.109,-57.703,174.437,19.037,153.125
C09963=1085.047,2.359,-57.718,174.438,19.039,153.125
C09964=1085.053,2.609,-57.732,174.440,19.041,153.125
C09965=1085.058,2.858,-57.746,174.441,19.043,153.125
C09966=1085.064,3.108,-57.759,174.443,19.045,153.125
C09967=1085.070,3.357,-57.773,174.444,19.047,153.125
C09968=1085.076,3.607,-57.788,174.446,19.049,153.125
C09969=1085.082,3.856,-57.802,174.448,19.051,153.126
C09970=1085.087,4.106,-57.815,174.449,19.053,153.126
C09971=1085.093,4.355,-57.829,174.451,19.055,153.126
C09972=1085.099,4.605,-57.843,174.452,19.057,153.126
C09973=1085.105,4.854,-57.858,174.454,19.059,153.126
C09974=1085.111,5.104,-57.871,174.455,19.061,153.126
C09975=1085.116,5.354,-57.885,174.457,19.063,153.126
C09976=1085.122,5.604,-57.899,174.458,19.065,153.126
C09977=1085.128,5.853,-57.914,174.460,19.067,153.126
C09978=1085.133,6.102,-57.928,174.461,19.068,153.127
C09979=1085.140,6.352,-57.941,174.463,19.071,153.127
C09980=1085.146,6.601,-57.956,174.464,19.072,153.127
C09981=1085.151,6.851,-57.970,174.466,19.074,153.127
C09982=1085.157,7.100,-57.984,174.468,19.076,153.127
C09983=1085.163,7.349,-57.998,174.469,19.078,153.127
C09984=1085.169,7.600,-58.013,174.470,19.080,153.127
C09985=1085.174,7.849,-58.027,174.472,19.082,153.127
C09986=1085.180,8.098,-58.041,174.474,19.085,153.127
C09987=1085.186,8.348,-58.055,174.475,19.086,153.127
C09988=1085.192,8.598,-58.069,174.476,19.088,153.128
C09989=1085.198,8.847,-58.083,174.479,19.090,153.128
C09990=1085.204,9.096,-58.097,174.480,19.092,153.128
C09991=1085.210,9.347,-58.111,174.481,19.094,153.128
C09992=1085.216,9.595,-58.126,174.483,19.096,153.128
C09993=1085.221,9.845,-58.140,174.485,19.098,153.128
C09994=1085.227,10.095,-58.155,174.486,19.100,153.128
C09995=1085.233,10.344,-58.169,174.488,19.101,153.128
C09996=1085.238,10.594,-58.182,174.490,19.104,153.128
//INST
///DATE 2021/06/17 10:54
///ATTR SC,RW,RJ
////FRAME ROBOT
///GROUP1 RB1
NOP
MOVL C00000 V=800.0 PL=0
MOVL C00001 V=800.0 PL=0
MOVL C00002 V=800.0 PL=0
MOVL C00003 V=800.0 PL=0
MOVL C00004 V=800.0 PL=0
MOVL C00005 V=800.0 PL=0
MOVL C00006 V=800.0 PL=0
MOVL C00007 V=800.0 PL=0
MOVL C00008 V=800.0 PL=0
MOVL C00009 V=800.0 PL=0
MOVL C00010 V=800.0 PL=0
MOVL C00011 V=800.0 PL=0
MOVL C00012 V=800.0 PL=0
MOVL C00013 V=800.0 PL=0
MOVL C00014 V=800.0 PL=0
MOVL C00015 V=800.0 PL=0
MOVL C00016 V=800.0 PL=0
MOVL C00017 V=800.0 PL=0
MOVL C00018 V=800.0 PL=0
MOVL C00019 V=800.0 PL=0
MOVL C00020 V=800.0 PL=0
MOVL C00021 V=800.0 PL=0
MOVL C00022 V=800.0 PL=0
MOVL C00023 V=800.0 PL=0
MOVL C00024 V=800.0 PL=0
MOVL C00025 V=800.0 PL=0
MOVL C00026 V=800.0 PL=0
MOVL C00027 V=800.0 PL=0
MOVL C00028 V=800.0 PL=0
MOVL C00029 V=800.0 PL=0
MOVL C00030 V=800.0 PL=0
MOVL C00031 V=800.0 PL=0
MOVL C00032 V=800.0 PL=0
MOVL C00033 V=800.0 PL=0
MOVL C00034 V=800.0 PL=0
MOVL C00035 V=800.0 PL=0
MOVL C00036 V=800.0 PL=0
MOVL C00037 V=800.0 PL=0
MOVL C00038 V=800.0 PL=0
MOVL C00039 V=800.0 PL=0
MOVL C00040 V=800.0 PL=0
MOVL C00041 V=800.0 PL=0
MOVL C00042 V=800.0 PL=0
MOVL C00043 V=800.0 PL=0
MOVL C00044 V=800.0 PL=0
MOVL C00045 V=800.0 PL=0
MOVL C00046 V=800.0 PL=0
MOVL C00047 V=800.0 PL=0
MOVL C00048 V=800.0 PL=0
MOVL C00049 V=800.0 PL=0
MOVL C00050 V=800.0 PL=0
MOVL C00051 V=800.0 PL=0
MOVL C00052 V=800.0 PL=0
MOVL C00053 V=800.0 PL=0
MOVL C00054 V=800.0 PL=0
MOVL C00055 V=800.0 PL=0
MOVL C00056 V=800.0 PL=0
MOVL C00057 V=800.0 PL=0
MOVL C00058 V=800.0 PL=0
MOVL C00059 V=800.0 PL=0
MOVL C00060 V=800.0 PL=0
MOVL C00061 V=800.0 PL=0
MOVL C00062 V=800.0 PL=0
MOVL C00063 V=800.0 PL=0
MOVL C00064 V=800.0 PL=0
MOVL C00065 V=800.0 PL=0
MOVL C00066 V=800.0 PL=0
MOVL C00067 V=800.0 PL=0
MOVL C00068 V=800.0 PL=0
MOVL C00069 V=800.0 PL=0
MOVL C00070 V=800.0 PL=0
MOVL C00071 V=800.0 PL=0
MOVL C00072 V=800.0 PL=0
MOVL C00073 V=800.0 PL=0
MOVL C00074 V=800.0 PL=0
MOVL C00075 V=800.0 PL=0
MOVL C00076 V=800.0 PL=0
MOVL C00077 V=800.0 PL=0
MOVL C00078 V=800.0 PL=0
MOVL C00079 V=800.0 PL=0
MOVL C00080 V=800.0 PL=0
MOVL C00081 V=800.0 PL=0
MOVL C00082 V=800.0 PL=0
MOVL C00083 V=800.0 PL=0
MOVL C00084 V=800.0 PL=0
MOVL C00085 V=800.0 PL=0
MOVL C00086 V=800.0 PL=0
MOVL C00087 V=800.0 PL=0
MOVL C00088 V=800.0 PL=0
MOVL C00089 V=800.0 PL=0
MOVL C00090 V=800.0 PL=0
MOVL C00091 V=800.0 PL=0
MOVL C00092 V=800.0 PL=0
MOVL C00093 V=800.0 PL=0
MOVL C00094 V=800.0 PL=0
MOVL C00095 V=800.0 PL=0
MOVL C00096 V=800.0 PL=0
MOVL C00097 V=800.0 PL=0
MOVL C00098 V=800.0 PL=0
MOVL C00099 V=800.0 PL=0
MOVL C00100 V=800.0 PL=0
MOVL C00101 V=800.0 PL=0
MOVL C00102 V=800.0 PL=0
MOVL C00103 V=800.0 PL=0
MOVL C00104 V=800.0 PL=0
MOVL C00105 V=800.0 PL=0
MOVL C00106 V=800.0 PL=0
MOVL C00107 V=800.0 PL=0
MOVL C00108 V=800.0 PL=0
MOVL C00109 V=800.0 PL=0
MOVL C00110 V=800.0 PL=0
MOVL C00111 V=800.0 PL=0
MOVL C00112 V=800.0 PL=0
MOVL C00113 V=800.0 PL=0
MOVL C00114 V=800.0 PL=0
MOVL C00115 V=800.0 PL=0
MOVL C00116 V=800.0 PL=0
MOVL C00117 V=800.0 PL=0
MOVL C00118 V=800.0 PL=0
MOVL C00119 V=800.0 PL=0
MOVL C00120 V=800.0 PL=0
MOVL C00121 V=800.0 PL=0
MOVL C00122 V=800.0 PL=0
MOVL C00123 V=800.0 PL=0
MOVL C00124 V=800.0 PL=0
MOVL C00125 V=800.0 PL=0
MOVL C00126 V=800.0 PL=0
MOVL C00127 V=800.0 PL=0
MOVL C00128 V=800.0 PL=0
MOVL C00129 V=800.0 PL=0
MOVL C00130 V=800.0 PL=0
MOVL C00131 V=800.0 PL=0
MOVL C00132 V=800.0 PL=0
MOVL C00133 V=800.0 PL=0
MOVL C00134 V=800.0 PL=0
MOVL C00135 V=800.0 PL=0
MOVL C00136 V=800.0 PL=0
MOVL C00137 V=800.0 PL=0
MOVL C00138 V=800.0 PL=0
MOVL C00139 V=800.0 PL=0
MOVL C00140 V=800.0 PL=0
MOVL C00141 V=800.0 PL=0
MOVL C00142 V=800.0 PL=0
MOVL C00143 V=800.0 PL=0
MOVL C00144 V=800.0 PL=0
MOVL C00145 V=800.0 PL=0
MOVL C00146 V=800.0 PL=0
MOVL C00147 V=800.0 PL=0
MOVL C00148 V=800.0 PL=0
MOVL C00149 V=800.0 PL=0
MOVL C00150 V=800.0 PL=0
MOVL C00151 V=800.0 PL=0
MOVL C00152 V=800.0 PL=0
MOVL C00153 V=800.0 PL=0
MOVL C00154 V=800.0 PL=0
MOVL C00155 V=800.0 PL=0
MOVL C00156 V=800.0 PL=0
MOVL C00157 V=800.0 PL=0
MOVL C00158 V=800.0 PL=0
MOVL C00159 V=800.0 PL=0
MOVL C00160 V=800.0 PL=0
MOVL C00161 V=800.0 PL=0
MOVL C00162 V=800.0 PL=0
MOVL C00163 V=800.0 PL=0
MOVL C00164 V=800.0 PL=0
MOVL C00165 V=800.0 PL=0
MOVL C00166 V=800.0 PL=0
MOVL C00167 V=800.0 PL=0
MOVL C00168 V=800.0 PL=0
MOVL C00169 V=800.0 PL=0
MOVL C00170 V=800.0 PL=0
MOVL C00171 V=800.0 PL=0
MOVL C00172 V=800.0 PL=0
MOVL C00173 V=800.0 PL=0
MOVL C00174 V=800.0 PL=0
MOVL C00175 V=800.0 PL=0
MOVL C00176 V=800.0 PL=0
MOVL C00177 V=800.0 PL=0
MOVL C00178 V=800.0 PL=0
MOVL C00179 V=800.0 PL=0
MOVL C00180 V=800.0 PL=0
MOVL C00181 V=800.0 PL=0
MOVL C00182 V=800.0 PL=0
MOVL C00183 V=800.0 PL=0
MOVL C00184 V=800.0 PL=0
MOVL C00185 V=800.0 PL=0
MOVL C00186 V=800.0 PL=0
MOVL C00187 V=800.0 PL=0
MOVL C00188 V=800.0 PL=0
MOVL C00189 V=800.0 PL=0
MOVL C00190 V=800.0 PL=0
MOVL C00191 V=800.0 PL=0
MOVL C00192 V=800.0 PL=0
MOVL C00193 V=800.0 PL=0
MOVL C00194 V=800.0 PL=0
MOVL C00195 V=800.0 PL=0
MOVL C00196 V=800.0 PL=0
MOVL C00197 V=800.0 PL=0
MOVL C00198 V=800.0 PL=0
MOVL C00199 V=800.0 PL=0
MOVL C00200 V=800.0 PL=0
MOVL C00201 V=800.0 PL=0
MOVL C00202 V=800.0 PL=0
MOVL C00203 V=800.0 PL=0
MOVL C00204 V=800.0 PL=0
MOVL C00205 V=800.0 PL=0
MOVL C00206 V=800.0 PL=0
MOVL C00207 V=800.0 PL=0
MOVL C00208 V=800.0 PL=0
MOVL C00209 V=800.0 PL=0
MOVL C00210 V=800.0 PL=0
MOVL C00211 V=800.0 PL=0
MOVL C00212 V=800.0 PL=0
MOVL C00213 V=800.0 PL=0
MOVL C00214 V=800.0 PL=0
MOVL C00215 V=800.0 PL=0
MOVL C00216 V=800.0 PL=0
MOVL C00217 V=800.0 PL=0
MOVL C00218 V=800.0 PL=0
MOVL C00219 V=800.0 PL=0
MOVL C00220 V=800.0 PL=0
MOVL C00221 V=800.0 PL=0
MOVL C00222 V=800.0 PL=0
MOVL C00223 V=800.0 PL=0
MOVL C00224 V=800.0 PL=0
MOVL C00225 V=800.0 PL=0
MOVL C00226 V=800.0 PL=0
MOVL C00227 V=800.0 PL=0
MOVL C00228 V=800.0 PL=0
MOVL C00229 V=800.0 PL=0
MOVL C00230 V=800.0 PL=0
MOVL C00231 V=800.0 PL=0
MOVL C00232 V=800.0 PL=0
MOVL C00233 V=800.0 PL=0
MOVL C00234 V=800.0 PL=0
MOVL C00235 V=800.0 PL=0
MOVL C00236 V=800.0 PL=0
MOVL C00237 V=800.0 PL=0
MOVL C00238 V=800.0 PL=0
MOVL C00239 V=800.0 PL=0
MOVL C00240 V=800.0 PL=0
MOVL C00241 V=800.0 PL=0
MOVL C00242 V=800.0 PL=0
MOVL C00243 V=800.0 PL=0
MOVL C00244 V=800.0 PL=0
MOVL C00245 V=800.0 PL=0
MOVL C00246 V=800.0 PL=0
MOVL C00247 V=800.0 PL=0
MOVL C00248 V=800.0 PL=0
MOVL C00249 V=800.0 PL=0
MOVL C00250 V=800.0 PL=0
MOVL C00251 V=800.0 PL=0
MOVL C00252 V=800.0 PL=0
MOVL C00253 V=800.0 PL=0
MOVL C00254 V=800.0 PL=0
MOVL C00255 V=800.0 PL=0
MOVL C00256 V=800.0 PL=0
MOVL C00257 V=800.0 PL=0
MOVL C00258 V=800.0 PL=0
MOVL C00259 V=800.0 PL=0
MOVL C00260 V=800.0 PL=0
MOVL C00261 V=800.0 PL=0
MOVL C00262 V=800.0 PL=0
MOVL C00263 V=800.0 PL=0
MOVL C00264 V=800.0 PL=0
MOVL C00265 V=800.0 PL=0
MOVL C00266 V=800.0 PL=0
MOVL C00267 V=800.0 PL=0
MOVL C00268 V=800.0 PL=0
MOVL C00269 V=800.0 PL=0
MOVL C00270 V=800.0 PL=0
MOVL C00271 V=800.0 PL=0
MOVL C00272 V=800.0 PL=0
MOVL C00273 V=800.0 PL=0
MOVL C00274 V=800.0 PL=0
MOVL C00275 V=800.0 PL=0
MOVL C00276 V=800.0 PL=0
MOVL C00277 V=800.0 PL=0
MOVL C00278 V=800.0 PL=0
MOVL C00279 V=800.0 PL=0
MOVL C00280 V=800.0 PL=0
MOVL C00281 V=800.0 PL=0
MOVL C00282 V=800.0 PL=0
MOVL C00283 V=800.0 PL=0
MOVL C00284 V=800.0 PL=0
MOVL C00285 V=800.0 PL=0
MOVL C00286 V=800.0 PL=0
MOVL C00287 V=800.0 PL=0
MOVL C00288 V=800.0 PL=0
MOVL C00289 V=800.0 PL=0
MOVL C00290 V=800.0 PL=0
MOVL C00291 V=800.0 PL=0
MOVL C00292 V=800.0 PL=0
MOVL C00293 V=800.0 PL=0
MOVL C00294 V=800.0 PL=0
MOVL C00295 V=800.0 PL=0
MOVL C00296 V=800.0 PL=0
MOVL C00297 V=800.0 PL=0
MOVL C00298 V=800.0 PL=0
MOVL C00299 V=800.0 PL=0
MOVL C00300 V=800.0 PL=0
MOVL C00301 V=800.0 PL=0
MOVL C00302 V=800.0 PL=0
MOVL C00303 V=800.0 PL=0
MOVL C00304 V=800.0 PL=0
MOVL C00305 V=800.0 PL=0
MOVL C00306 V=800.0 PL=0
MOVL C00307 V=800.0 PL=0
MOVL C00308 V=800.0 PL=0
MOVL C00309 V=800.0 PL=0
MOVL C00310 V=800.0 PL=0
MOVL C00311 V=800.0 PL=0
MOVL C00312 V=800.0 PL=0
MOVL C00313 V=800.0 PL=0
MOVL C00314 V=800.0 PL=0
MOVL C00315 V=800.0 PL=0
MOVL C00316 V=800.0 PL=0
MOVL C00317 V=800.0 PL=0
MOVL C00318 V=800.0 PL=0
MOVL C00319 V=800.0 PL=0
MOVL C00320 V=800.0 PL=0
MOVL C00321 V=800.0 PL=0
MOVL C00322 V=800.0 PL=0
MOVL C00323 V=800.0 PL=0
MOVL C00324 V=800.0 PL=0
MOVL C00325 V=800.0 PL=0
MOVL C00326 V=800.0 PL=0
MOVL C00327 V=800.0 PL=0
MOVL C00328 V=800.0 PL=0
MOVL C00329 V=800.0 PL=0
MOVL C00330 V=800.0 PL=0
MOVL C00331 V=800.0 PL=0
MOVL C00332 V=800.0 PL=0
MOVL C00333 V=800.0 PL=0
MOVL C00334 V=800.0 PL=0
MOVL C00335 V=800.0 PL=0
MOVL C00336 V=800.0 PL=0
MOVL C00337 V=800.0 PL=0
MOVL C00338 V=800.0 PL=0
MOVL C00339 V=800.0 PL=0
MOVL C00340 V=800.0 PL=0
MOVL C00341 V=800.0 PL=0
MOVL C00342 V=800.0 PL=0
MOVL C00343 V=800.0 PL=0
MOVL C00344 V=800.0 PL=0
MOVL C00345 V=800.0 PL=0
MOVL C00346 V=800.0 PL=0
MOVL C00347 V=800.0 PL=0
MOVL C00348 V=800.0 PL=0
MOVL C00349 V=800.0 PL=0
MOVL C00350 V=800.0 PL=0
MOVL C00351 V=800.0 PL=0
MOVL C00352 V=800.0 PL=0
MOVL C00353 V=800.0 PL=0
MOVL C00354 V=800.0 PL=0
MOVL C00355 V=800.0 PL=0
MOVL C00356 V=800.0 PL=0
MOVL C00357 V=800.0 PL=0
MOVL C00358 V=800.0 PL=0
MOVL C00359 V=800.0 PL=0
MOVL C00360 V=800.0 PL=0
MOVL C00361 V=800.0 PL=0
MOVL C00362 V=800.0 PL=0
MOVL C00363 V=800.0 PL=0
MOVL C00364 V=800.0 PL=0
MOVL C00365 V=800.0 PL=0
MOVL C00366 V=800.0 PL=0
MOVL C00367 V=800.0 PL=0
MOVL C00368 V=800.0 PL=0
MOVL C00369 V=800.0 PL=0
MOVL C00370 V=800.0 PL=0
MOVL C00371 V=800.0 PL=0
MOVL C00372 V=800.0 PL=0
MOVL C00373 V=800.0 PL=0
MOVL C00374 V=800.0 PL=0
MOVL C00375 V=800.0 PL=0
MOVL C00376 V=800.0 PL=0
MOVL C00377 V=800.0 PL=0
MOVL C00378 V=800.0 PL=0
MOVL C00379 V=800.0 PL=0
MOVL C00380 V=800.0 PL=0
MOVL C00381 V=800.0 PL=0
MOVL C00382 V=800.0 PL=0
MOVL C00383 V=800.0 PL=0
MOVL C00384 V=800.0 PL=0
MOVL C00385 V=800.0 PL=0
MOVL C00386 V=800.0 PL=0
MOVL C00387 V=800.0 PL=0
MOVL C00388 V=800.0 PL=0
MOVL C00389 V=800.0 PL=0
MOVL C00390 V=800.0 PL=0
MOVL C00391 V=800.0 PL=0
MOVL C00392 V=800.0 PL=0
MOVL C00393 V=800.0 PL=0
MOVL C00394 V=800.0 PL=0
MOVL C00395 V=800.0 PL=0
MOVL C00396 V=800.0 PL=0
MOVL C00397 V=800.0 PL=0
MOVL C00398 V=800.0 PL=0
MOVL C00399 V=800.0 PL=0
MOVL C00400 V=800.0 PL=0
MOVL C00401 V=800.0 PL=0
MOVL C00402 V=800.0 PL=0
MOVL C00403 V=800.0 PL=0
MOVL C00404 V=800.0 PL=0
MOVL C00405 V=800.0 PL=0
MOVL C00406 V=800.0 PL=0
MOVL C00407 V=800.0 PL=0
MOVL C00408 V=800.0 PL=0
MOVL C00409 V=800.0 PL=0
MOVL C00410 V=800.0 PL=0
MOVL C00411 V=800.0 PL=0
MOVL C00412 V=800.0 PL=0
MOVL C00413 V=800.0 PL=0
MOVL C00414 V=800.0 PL=0
MOVL C00415 V=800.0 PL=0
MOVL C00416 V=800.0 PL=0
MOVL C00417 V=800.0 PL=0
MOVL C00418 V=800.0 PL=0
MOVL C00419 V=800.0 PL=0
MOVL C00420 V=800.0 PL=0
MOVL C00421 V=800.0 PL=0
MOVL C00422 V=800.0 PL=0
MOVL C00423 V=800.0 PL=0
MOVL C00424 V=800.0 PL=0
MOVL C00425 V=800.0 PL=0
MOVL C00426 V=800.0 PL=0
MOVL C00427 V=800.0 PL=0
MOVL C00428 V=800.0 PL=0
MOVL C00429 V=800.0 PL=0
MOVL C00430 V=800.0 PL=0
MOVL C00431 V=800.0 PL=0
MOVL C00432 V=800.0 PL=0
MOVL C00433 V=800.0 PL=0
MOVL C00434 V=800.0 PL=0
MOVL C00435 V=800.0 PL=0
MOVL C00436 V=800.0 PL=0
MOVL C00437 V=800.0 PL=0
MOVL C00438 V=800.0 PL=0
MOVL C00439 V=800.0 PL=0
MOVL C00440 V=800.0 PL=0
MOVL C00441 V=800.0 PL=0
MOVL C00442 V=800.0 PL=0
MOVL C00443 V=800.0 PL=0
MOVL C00444 V=800.0 PL=0
MOVL C00445 V=800.0 PL=0
MOVL C00446 V=800.0 PL=0
MOVL C00447 V=800.0 PL=0
MOVL C00448 V=800.0 PL=0
MOVL C00449 V=800.0 PL=0
MOVL C00450 V=800.0 PL=0
MOVL C00451 V=800.0 PL=0
MOVL C00452 V=800.0 PL=0
MOVL C00453 V=800.0 PL=0
MOVL C00454 V=800.0 PL=0
MOVL C00455 V=800.0 PL=0
MOVL C00456 V=800.0 PL=0
MOVL C00457 V=800.0 PL=0
MOVL C00458 V=800.0 PL=0
MOVL C00459 V=800.0 PL=0
MOVL C00460 V=800.0 PL=0
MOVL C00461 V=800.0 PL=0
MOVL C00462 V=800.0 PL=0
MOVL C00463 V=800.0 PL=0
MOVL C00464 V=800.0 PL=0
MOVL C00465 V=800.0 PL=0
MOVL C00466 V=800.0 PL=0
MOVL C00467 V=800.0 PL=0
MOVL C00468 V=800.0 PL=0
MOVL C00469 V=800.0 PL=0
MOVL C00470 V=800.0 PL=0
MOVL C00471 V=800.0 PL=0
MOVL C00472 V=800.0 PL=0
MOVL C00473 V=800.0 PL=0
MOVL C00474 V=800.0 PL=0
MOVL C00475 V=800.0 PL=0
MOVL C00476 V=800.0 PL=0
MOVL C00477 V=800.0 PL=0
MOVL C00478 V=800.0 PL=0
MOVL C00479 V=800.0 PL=0
MOVL C00480 V=800.0 PL=0
MOVL C00481 V=800.0 PL=0
MOVL C00482 V=800.0 PL=0
MOVL C00483 V=800.0 PL=0
MOVL C00484 V=800.0 PL=0
MOVL C00485 V=800.0 PL=0
MOVL C00486 V=800.0 PL=0
MOVL C00487 V=800.0 PL=0
MOVL C00488 V=800.0 PL=0
MOVL C00489 V=800.0 PL=0
MOVL C00490 V=800.0 PL=0
MOVL C00491 V=800.0 PL=0
MOVL C00492 V=800.0 PL=0
MOVL C00493 V=800.0 PL=0
MOVL C00494 V=800.0 PL=0
MOVL C00495 V=800.0 PL=0
MOVL C00496 V=800.0 PL=0
MOVL C00497 V=800.0 PL=0
MOVL C00498 V=800.0 PL=0
MOVL C00499 V=800.0 PL=0
MOVL C00500 V=800.0 PL=0
MOVL C00501 V=800.0 PL=0
MOVL C00502 V=800.0 PL=0
MOVL C00503 V=800.0 PL=0
MOVL C00504 V=800.0 PL=0
MOVL C00505 V=800.0 PL=0
MOVL C00506 V=800.0 PL=0
MOVL C00507 V=800.0 PL=0
MOVL C00508 V=800.0 PL=0
MOVL C00509 V=800.0 PL=0
MOVL C00510 V=800.0 PL=0
MOVL C00511 V=800.0 PL=0
MOVL C00512 V=800.0 PL=0
MOVL C00513 V=800.0 PL=0
MOVL C00514 V=800.0 PL=0
MOVL C00515 V=800.0 PL=0
MOVL C00516 V=800.0 PL=0
MOVL C00517 V=800.0 PL=0
MOVL C00518 V=800.0 PL=0
MOVL C00519 V=800.0 PL=0
MOVL C00520 V=800.0 PL=0
MOVL C00521 V=800.0 PL=0
MOVL C00522 V=800.0 PL=0
MOVL C00523 V=800.0 PL=0
MOVL C00524 V=800.0 PL=0
MOVL C00525 V=800.0 PL=0
MOVL C00526 V=800.0 PL=0
MOVL C00527 V=800.0 PL=0
MOVL C00528 V=800.0 PL=0
MOVL C00529 V=800.0 PL=0
MOVL C00530 V=800.0 PL=0
MOVL C00531 V=800.0 PL=0
MOVL C00532 V=800.0 PL=0
MOVL C00533 V=800.0 PL=0
MOVL C00534 V=800.0 PL=0
MOVL C00535 V=800.0 PL=0
MOVL C00536 V=800.0 PL=0
MOVL C00537 V=800.0 PL=0
MOVL C00538 V=800.0 PL=0
MOVL C00539 V=800.0 PL=0
MOVL C00540 V=800.0 PL=0
MOVL C00541 V=800.0 PL=0
MOVL C00542 V=800.0 PL=0
MOVL C00543 V=800.0 PL=0
MOVL C00544 V=800.0 PL=0
MOVL C00545 V=800.0 PL=0
MOVL C00546 V=800.0 PL=0
MOVL C00547 V=800.0 PL=0
MOVL C00548 V=800.0 PL=0
MOVL C00549 V=800.0 PL=0
MOVL C00550 V=800.0 PL=0
MOVL C00551 V=800.0 PL=0
MOVL C00552 V=800.0 PL=0
MOVL C00553 V=800.0 PL=0
MOVL C00554 V=800.0 PL=0
MOVL C00555 V=800.0 PL=0
MOVL C00556 V=800.0 PL=0
MOVL C00557 V=800.0 PL=0
MOVL C00558 V=800.0 PL=0
MOVL C00559 V=800.0 PL=0
MOVL C00560 V=800.0 PL=0
MOVL C00561 V=800.0 PL=0
MOVL C00562 V=800.0 PL=0
MOVL C00563 V=800.0 PL=0
MOVL C00564 V=800.0 PL=0
MOVL C00565 V=800.0 PL=0
MOVL C00566 V=800.0 PL=0
MOVL C00567 V=800.0 PL=0
MOVL C00568 V=800.0 PL=0
MOVL C00569 V=800.0 PL=0
MOVL C00570 V=800.0 PL=0
MOVL C00571 V=800.0 PL=0
MOVL C00572 V=800.0 PL=0
MOVL C00573 V=800.0 PL=0
MOVL C00574 V=800.0 PL=0
MOVL C00575 V=800.0 PL=0
MOVL C00576 V=800.0 PL=0
MOVL C00577 V=800.0 PL=0
MOVL C00578 V=800.0 PL=0
MOVL C00579 V=800.0 PL=0
MOVL C00580 V=800.0 PL=0
MOVL C00581 V=800.0 PL=0
MOVL C00582 V=800.0 PL=0
MOVL C00583 V=800.0 PL=0
MOVL C00584 V=800.0 PL=0
MOVL C00585 V=800.0 PL=0
MOVL C00586 V=800.0 PL=0
MOVL C00587 V=800.0 PL=0
MOVL C00588 V=800.0 PL=0
MOVL C00589 V=800.0 PL=0
MOVL C00590 V=800.0 PL=0
MOVL C00591 V=800.0 PL=0
MOVL C00592 V=800.0 PL=0
MOVL C00593 V=800.0 PL=0
MOVL C00594 V=800.0 PL=0
MOVL C00595 V=800.0 PL=0
MOVL C00596 V=800.0 PL=0
MOVL C00597 V=800.0 PL=0
MOVL C00598 V=800.0 PL=0
MOVL C00599 V=800.0 PL=0
MOVL C00600 V=800.0 PL=0
MOVL C00601 V=800.0 PL=0
MOVL C00602 V=800.0 PL=0
MOVL C00603 V=800.0 PL=0
MOVL C00604 V=800.0 PL=0
MOVL C00605 V=800.0 PL=0
MOVL C00606 V=800.0 PL=0
MOVL C00607 V=800.0 PL=0
MOVL C00608 V=800.0 PL=0
MOVL C00609 V=800.0 PL=0
MOVL C00610 V=800.0 PL=0
MOVL C00611 V=800.0 PL=0
MOVL C00612 V=800.0 PL=0
MOVL C00613 V=800.0 PL=0
MOVL C00614 V=800.0 PL=0
MOVL C00615 V=800.0 PL=0
MOVL C00616 V=800.0 PL=0
MOVL C00617 V=800.0 PL=0
MOVL C00618 V=800.0 PL=0
MOVL C00619 V=800.0 PL=0
MOVL C00620 V=800.0 PL=0
MOVL C00621 V=800.0 PL=0
MOVL C00622 V=800.0 PL=0
MOVL C00623 V=800.0 PL=0
MOVL C00624 V=800.0 PL=0
MOVL C00625 V=800.0 PL=0
MOVL C00626 V=800.0 PL=0
MOVL C00627 V=800.0 PL=0
MOVL C00628 V=800.0 PL=0
MOVL C00629 V=800.0 PL=0
MOVL C00630 V=800.0 PL=0
MOVL C00631 V=800.0 PL=0
MOVL C00632 V=800.0 PL=0
MOVL C00633 V=800.0 PL=0
MOVL C00634 V=800.0 PL=0
MOVL C00635 V=800.0 PL=0
MOVL C00636 V=800.0 PL=0
MOVL C00637 V=800.0 PL=0
MOVL C00638 V=800.0 PL=0
MOVL C00639 V=800.0 PL=0
MOVL C00640 V=800.0 PL=0
MOVL C00641 V=800.0 PL=0
MOVL C00642 V=800.0 PL=0
MOVL C00643 V=800.0 PL=0
MOVL C00644 V=800.0 PL=0
MOVL C00645 V=800.0 PL=0
MOVL C00646 V=800.0 PL=0
MOVL C00647 V=800.0 PL=0
MOVL C00648 V=800.0 PL=0
MOVL C00649 V=800.0 PL=0
MOVL C00650 V=800.0 PL=0
MOVL C00651 V=800.0 PL=0
MOVL C00652 V=800.0 PL=0
MOVL C00653 V=800.0 PL=0
MOVL C00654 V=800.0 PL=0
MOVL C00655 V=800.0 PL=0
MOVL C00656 V=800.0 PL=0
MOVL C00657 V=800.0 PL=0
MOVL C00658 V=800.0 PL=0
MOVL C00659 V=800.0 PL=0
MOVL C00660 V=800.0 PL=0
MOVL C00661 V=800.0 PL=0
MOVL C00662 V=800.0 PL=0
MOVL C00663 V=800.0 PL=0
MOVL C00664 V=800.0 PL=0
MOVL C00665 V=800.0 PL=0
MOVL C00666 V=800.0 PL=0
MOVL C00667 V=800.0 PL=0
MOVL C00668 V=800.0 PL=0
MOVL C00669 V=800.0 PL=0
MOVL C00670 V=800.0 PL=0
MOVL C00671 V=800.0 PL=0
MOVL C00672 V=800.0 PL=0
MOVL C00673 V=800.0 PL=0
MOVL C00674 V=800.0 PL=0
MOVL C00675 V=800.0 PL=0
MOVL C00676 V=800.0 PL=0
MOVL C00677 V=800.0 PL=0
MOVL C00678 V=800.0 PL=0
MOVL C00679 V=800.0 PL=0
MOVL C00680 V=800.0 PL=0
MOVL C00681 V=800.0 PL=0
MOVL C00682 V=800.0 PL=0
MOVL C00683 V=800.0 PL=0
MOVL C00684 V=800.0 PL=0
MOVL C00685 V=800.0 PL=0
MOVL C00686 V=800.0 PL=0
MOVL C00687 V=800.0 PL=0
MOVL C00688 V=800.0 PL=0
MOVL C00689 V=800.0 PL=0
MOVL C00690 V=800.0 PL=0
MOVL C00691 V=800.0 PL=0
MOVL C00692 V=800.0 PL=0
MOVL C00693 V=800.0 PL=0
MOVL C00694 V=800.0 PL=0
MOVL C00695 V=800.0 PL=0
MOVL C00696 V=800.0 PL=0
MOVL C00697 V=800.0 PL=0
MOVL C00698 V=800.0 PL=0
MOVL C00699 V=800.0 PL=0
MOVL C00700 V=800.0 PL=0
MOVL C00701 V=800.0 PL=0
MOVL C00702 V=800.0 PL=0
MOVL C00703 V=800.0 PL=0
MOVL C00704 V=800.0 PL=0
MOVL C00705 V=800.0 PL=0
MOVL C00706 V=800.0 PL=0
MOVL C00707 V=800.0 PL=0
MOVL C00708 V=800.0 PL=0
MOVL C00709 V=800.0 PL=0
MOVL C00710 V=800.0 PL=0
MOVL C00711 V=800.0 PL=0
MOVL C00712 V=800.0 PL=0
MOVL C00713 V=800.0 PL=0
MOVL C00714 V=800.0 PL=0
MOVL C00715 V=800.0 PL=0
MOVL C00716 V=800.0 PL=0
MOVL C00717 V=800.0 PL=0
MOVL C00718 V=800.0 PL=0
MOVL C00719 V=800.0 PL=0
MOVL C00720 V=800.0 PL=0
MOVL C00721 V=800.0 PL=0
MOVL C00722 V=800.0 PL=0
MOVL C00723 V=800.0 PL=0
MOVL C00724 V=800.0 PL=0
MOVL C00725 V=800.0 PL=0
MOVL C00726 V=800.0 PL=0
MOVL C00727 V=800.0 PL=0
MOVL C00728 V=800.0 PL=0
MOVL C00729 V=800.0 PL=0
MOVL C00730 V=800.0 PL=0
MOVL C00731 V=800.0 PL=0
MOVL C00732 V=800.0 PL=0
MOVL C00733 V=800.0 PL=0
MOVL C00734 V=800.0 PL=0
MOVL C00735 V=800.0 PL=0
MOVL C00736 V=800.0 PL=0
MOVL C00737 V=800.0 PL=0
MOVL C00738 V=800.0 PL=0
MOVL C00739 V=800.0 PL=0
MOVL C00740 V=800.0 PL=0
MOVL C00741 V=800.0 PL=0
MOVL C00742 V=800.0 PL=0
MOVL C00743 V=800.0 PL=0
MOVL C00744 V=800.0 PL=0
MOVL C00745 V=800.0 PL=0
MOVL C00746 V=800.0 PL=0
MOVL C00747 V=800.0 PL=0
MOVL C00748 V=800.0 PL=0
MOVL C00749 V=800.0 PL=0
MOVL C00750 V=800.0 PL=0
MOVL C00751 V=800.0 PL=0
MOVL C00752 V=800.0 PL=0
MOVL C00753 V=800.0 PL=0
MOVL C00754 V=800.0 PL=0
MOVL C00755 V=800.0 PL=0
MOVL C00756 V=800.0 PL=0
MOVL C00757 V=800.0 PL=0
MOVL C00758 V=800.0 PL=0
MOVL C00759 V=800.0 PL=0
MOVL C00760 V=800.0 PL=0
MOVL C00761 V=800.0 PL=0
MOVL C00762 V=800.0 PL=0
MOVL C00763 V=800.0 PL=0
MOVL C00764 V=800.0 PL=0
MOVL C00765 V=800.0 PL=0
MOVL C00766 V=800.0 PL=0
MOVL C00767 V=800.0 PL=0
MOVL C00768 V=800.0 PL=0
MOVL C00769 V=800.0 PL=0
MOVL C00770 V=800.0 PL=0
MOVL C00771 V=800.0 PL=0
MOVL C00772 V=800.0 PL=0
MOVL C00773 V=800.0 PL=0
MOVL C00774 V=800.0 PL=0
MOVL C00775 V=800.0 PL=0
MOVL C00776 V=800.0 PL=0
MOVL C00777 V=800.0 PL=0
MOVL C00778 V=800.0 PL=0
MOVL C00779 V=800.0 PL=0
MOVL C00780 V=800.0 PL=0
MOVL C00781 V=800.0 PL=0
MOVL C00782 V=800.0 PL=0
MOVL C00783 V=800.0 PL=0
MOVL C00784 V=800.0 PL=0
MOVL C00785 V=800.0 PL=0
MOVL C00786 V=800.0 PL=0
MOVL C00787 V=800.0 PL=0
MOVL C00788 V=800.0 PL=0
MOVL C00789 V=800.0 PL=0
MOVL C00790 V=800.0 PL=0
MOVL C00791 V=800.0 PL=0
MOVL C00792 V=800.0 PL=0
MOVL C00793 V=800.0 PL=0
MOVL C00794 V=800.0 PL=0
MOVL C00795 V=800.0 PL=0
MOVL C00796 V=800.0 PL=0
MOVL C00797 V=800.0 PL=0
MOVL C00798 V=800.0 PL=0
MOVL C00799 V=800.0 PL=0
MOVL C00800 V=800.0 PL=0
MOVL C00801 V=800.0 PL=0
MOVL C00802 V=800.0 PL=0
MOVL C00803 V=800.0 PL=0
MOVL C00804 V=800.0 PL=0
MOVL C00805 V=800.0 PL=0
MOVL C00806 V=800.0 PL=0
MOVL C00807 V=800.0 PL=0
MOVL C00808 V=800.0 PL=0
MOVL C00809 V=800.0 PL=0
MOVL C00810 V=800.0 PL=0
MOVL C00811 V=800.0 PL=0
MOVL C00812 V=800.0 PL=0
MOVL C00813 V=800.0 PL=0
MOVL C00814 V=800.0 PL=0
MOVL C00815 V=800.0 PL=0
MOVL C00816 V=800.0 PL=0
MOVL C00817 V=800.0 PL=0
MOVL C00818 V=800.0 PL=0
MOVL C00819 V=800.0 PL=0
MOVL C00820 V=800.0 PL=0
MOVL C00821 V=800.0 PL=0
MOVL C00822 V=800.0 PL=0
MOVL C00823 V=800.0 PL=0
MOVL C00824 V=800.0 PL=0
MOVL C00825 V=800.0 PL=0
MOVL C00826 V=800.0 PL=0
MOVL C00827 V=800.0 PL=0
MOVL C00828 V=800.0 PL=0
MOVL C00829 V=800.0 PL=0
MOVL C00830 V=800.0 PL=0
MOVL C00831 V=800.0 PL=0
MOVL C00832 V=800.0 PL=0
MOVL C00833 V=800.0 PL=0
MOVL C00834 V=800.0 PL=0
MOVL C00835 V=800.0 PL=0
MOVL C00836 V=800.0 PL=0
MOVL C00837 V=800.0 PL=0
MOVL C00838 V=800.0 PL=0
MOVL C00839 V=800.0 PL=0
MOVL C00840 V=800.0 PL=0
MOVL C00841 V=800.0 PL=0
MOVL C00842 V=800.0 PL=0
MOVL C00843 V=800.0 PL=0
MOVL C00844 V=800.0 PL=0
MOVL C00845 V=800.0 PL=0
MOVL C00846 V=800.0 PL=0
MOVL C00847 V=800.0 PL=0
MOVL C00848 V=800.0 PL=0
MOVL C00849 V=800.0 PL=0
MOVL C00850 V=800.0 PL=0
MOVL C00851 V=800.0 PL=0
MOVL C00852 V=800.0 PL=0
MOVL C00853 V=800.0 PL=0
MOVL C00854 V=800.0 PL=0
MOVL C00855 V=800.0 PL=0
MOVL C00856 V=800.0 PL=0
MOVL C00857 V=800.0 PL=0
MOVL C00858 V=800.0 PL=0
MOVL C00859 V=800.0 PL=0
MOVL C00860 V=800.0 PL=0
MOVL C00861 V=800.0 PL=0
MOVL C00862 V=800.0 PL=0
MOVL C00863 V=800.0 PL=0
MOVL C00864 V=800.0 PL=0
MOVL C00865 V=800.0 PL=0
MOVL C00866 V=800.0 PL=0
MOVL C00867 V=800.0 PL=0
MOVL C00868 V=800.0 PL=0
MOVL C00869 V=800.0 PL=0
MOVL C00870 V=800.0 PL=0
MOVL C00871 V=800.0 PL=0
MOVL C00872 V=800.0 PL=0
MOVL C00873 V=800.0 PL=0
MOVL C00874 V=800.0 PL=0
MOVL C00875 V=800.0 PL=0
MOVL C00876 V=800.0 PL=0
MOVL C00877 V=800.0 PL=0
MOVL C00878 V=800.0 PL=0
MOVL C00879 V=800.0 PL=0
MOVL C00880 V=800.0 PL=0
MOVL C00881 V=800.0 PL=0
MOVL C00882 V=800.0 PL=0
MOVL C00883 V=800.0 PL=0
MOVL C00884 V=800.0 PL=0
MOVL C00885 V=800.0 PL=0
MOVL C00886 V=800.0 PL=0
MOVL C00887 V=800.0 PL=0
MOVL C00888 V=800.0 PL=0
MOVL C00889 V=800.0 PL=0
MOVL C00890 V=800.0 PL=0
MOVL C00891 V=800.0 PL=0
MOVL C00892 V=800.0 PL=0
MOVL C00893 V=800.0 PL=0
MOVL C00894 V=800.0 PL=0
MOVL C00895 V=800.0 PL=0
MOVL C00896 V=800.0 PL=0
MOVL C00897 V=800.0 PL=0
MOVL C00898 V=800.0 PL=0
MOVL C00899 V=800.0 PL=0
MOVL C00900 V=800.0 PL=0
MOVL C00901 V=800.0 PL=0
MOVL C00902 V=800.0 PL=0
MOVL C00903 V=800.0 PL=0
MOVL C00904 V=800.0 PL=0
MOVL C00905 V=800.0 PL=0
MOVL C00906 V=800.0 PL=0
MOVL C00907 V=800.0 PL=0
MOVL C00908 V=800.0 PL=0
MOVL C00909 V=800.0 PL=0
MOVL C00910 V=800.0 PL=0
MOVL C00911 V=800.0 PL=0
MOVL C00912 V=800.0 PL=0
MOVL C00913 V=800.0 PL=0
MOVL C00914 V=800.0 PL=0
MOVL C00915 V=800.0 PL=0
MOVL C00916 V=800.0 PL=0
MOVL C00917 V=800.0 PL=0
MOVL C00918 V=800.0 PL=0
MOVL C00919 V=800.0 PL=0
MOVL C00920 V=800.0 PL=0
MOVL C00921 V=800.0 PL=0
MOVL C00922 V=800.0 PL=0
MOVL C00923 V=800.0 PL=0
MOVL C00924 V=800.0 PL=0
MOVL C00925 V=800.0 PL=0
MOVL C00926 V=800.0 PL=0
MOVL C00927 V=800.0 PL=0
MOVL C00928 V=800.0 PL=0
MOVL C00929 V=800.0 PL=0
MOVL C00930 V=800.0 PL=0
MOVL C00931 V=800.0 PL=0
MOVL C00932 V=800.0 PL=0
MOVL C00933 V=800.0 PL=0
MOVL C00934 V=800.0 PL=0
MOVL C00935 V=800.0 PL=0
MOVL C00936 V=800.0 PL=0
MOVL C00937 V=800.0 PL=0
MOVL C00938 V=800.0 PL=0
MOVL C00939 V=800.0 PL=0
MOVL C00940 V=800.0 PL=0
MOVL C00941 V=800.0 PL=0
MOVL C00942 V=800.0 PL=0
MOVL C00943 V=800.0 PL=0
MOVL C00944 V=800.0 PL=0
MOVL C00945 V=800.0 PL=0
MOVL C00946 V=800.0 PL=0
MOVL C00947 V=800.0 PL=0
MOVL C00948 V=800.0 PL=0
MOVL C00949 V=800.0 PL=0
MOVL C00950 V=800.0 PL=0
MOVL C00951 V=800.0 PL=0
MOVL C00952 V=800.0 PL=0
MOVL C00953 V=800.0 PL=0
MOVL C00954 V=800.0 PL=0
MOVL C00955 V=800.0 PL=0
MOVL C00956 V=800.0 PL=0
MOVL C00957 V=800.0 PL=0
MOVL C00958 V=800.0 PL=0
MOVL C00959 V=800.0 PL=0
MOVL C00960 V=800.0 PL=0
MOVL C00961 V=800.0 PL=0
MOVL C00962 V=800.0 PL=0
MOVL C00963 V=800.0 PL=0
MOVL C00964 V=800.0 PL=0
MOVL C00965 V=800.0 PL=0
MOVL C00966 V=800.0 PL=0
MOVL C00967 V=800.0 PL=0
MOVL C00968 V=800.0 PL=0
MOVL C00969 V=800.0 PL=0
MOVL C00970 V=800.0 PL=0
MOVL C00971 V=800.0 PL=0
MOVL C00972 V=800.0 PL=0
MOVL C00973 V=800.0 PL=0
MOVL C00974 V=800.0 PL=0
MOVL C00975 V=800.0 PL=0
MOVL C00976 V=800.0 PL=0
MOVL C00977 V=800.0 PL=0
MOVL C00978 V=800.0 PL=0
MOVL C00979 V=800.0 PL=0
MOVL C00980 V=800.0 PL=0
MOVL C00981 V=800.0 PL=0
MOVL C00982 V=800.0 PL=0
MOVL C00983 V=800.0 PL=0
MOVL C00984 V=800.0 PL=0
MOVL C00985 V=800.0 PL=0
MOVL C00986 V=800.0 PL=0
MOVL C00987 V=800.0 PL=0
MOVL C00988 V=800.0 PL=0
MOVL C00989 V=800.0 PL=0
MOVL C00990 V=800.0 PL=0
MOVL C00991 V=800.0 PL=0
MOVL C00992 V=800.0 PL=0
MOVL C00993 V=800.0 PL=0
MOVL C00994 V=800.0 PL=0
MOVL C00995 V=800.0 PL=0
MOVL C00996 V=800.0 PL=0
MOVL C00997 V=800.0 PL=0
MOVL C00998 V=800.0 PL=0
MOVL C00999 V=800.0 PL=0
MOVL C01000 V=800.0 PL=0
MOVL C01001 V=800.0 PL=0
MOVL C01002 V=800.0 PL=0
MOVL C01003 V=800.0 PL=0
MOVL C01004 V=800.0 PL=0
MOVL C01005 V=800.0 PL=0
MOVL C01006 V=800.0 PL=0
MOVL C01007 V=800.0 PL=0
MOVL C01008 V=800.0 PL=0
MOVL C01009 V=800.0 PL=0
MOVL C01010 V=800.0 PL=0
MOVL C01011 V=800.0 PL=0
MOVL C01012 V=800.0 PL=0
MOVL C01013 V=800.0 PL=0
MOVL C01014 V=800.0 PL=0
MOVL C01015 V=800.0 PL=0
MOVL C01016 V=800.0 PL=0
MOVL C01017 V=800.0 PL=0
MOVL C01018 V=800.0 PL=0
MOVL C01019 V=800.0 PL=0
MOVL C01020 V=800.0 PL=0
MOVL C01021 V=800.0 PL=0
MOVL C01022 V=800.0 PL=0
MOVL C01023 V=800.0 PL=0
MOVL C01024 V=800.0 PL=0
MOVL C01025 V=800.0 PL=0
MOVL C01026 V=800.0 PL=0
MOVL C01027 V=800.0 PL=0
MOVL C01028 V=800.0 PL=0
MOVL C01029 V=800.0 PL=0
MOVL C01030 V=800.0 PL=0
MOVL C01031 V=800.0 PL=0
MOVL C01032 V=800.0 PL=0
MOVL C01033 V=800.0 PL=0
MOVL C01034 V=800.0 PL=0
MOVL C01035 V=800.0 PL=0
MOVL C01036 V=800.0 PL=0
MOVL C01037 V=800.0 PL=0
MOVL C01038 V=800.0 PL=0
MOVL C01039 V=800.0 PL=0
MOVL C01040 V=800.0 PL=0
MOVL C01041 V=800.0 PL=0
MOVL C01042 V=800.0 PL=0
MOVL C01043 V=800.0 PL=0
MOVL C01044 V=800.0 PL=0
MOVL C01045 V=800.0 PL=0
MOVL C01046 V=800.0 PL=0
MOVL C01047 V=800.0 PL=0
MOVL C01048 V=800.0 PL=0
MOVL C01049 V=800.0 PL=0
MOVL C01050 V=800.0 PL=0
MOVL C01051 V=800.0 PL=0
MOVL C01052 V=800.0 PL=0
MOVL C01053 V=800.0 PL=0
MOVL C01054 V=800.0 PL=0
MOVL C01055 V=800.0 PL=0
MOVL C01056 V=800.0 PL=0
MOVL C01057 V=800.0 PL=0
MOVL C01058 V=800.0 PL=0
MOVL C01059 V=800.0 PL=0
MOVL C01060 V=800.0 PL=0
MOVL C01061 V=800.0 PL=0
MOVL C01062 V=800.0 PL=0
MOVL C01063 V=800.0 PL=0
MOVL C01064 V=800.0 PL=0
MOVL C01065 V=800.0 PL=0
MOVL C01066 V=800.0 PL=0
MOVL C01067 V=800.0 PL=0
MOVL C01068 V=800.0 PL=0
MOVL C01069 V=800.0 PL=0
MOVL C01070 V=800.0 PL=0
MOVL C01071 V=800.0 PL=0
MOVL C01072 V=800.0 PL=0
MOVL C01073 V=800.0 PL=0
MOVL C01074 V=800.0 PL=0
MOVL C01075 V=800.0 PL=0
MOVL C01076 V=800.0 PL=0
MOVL C01077 V=800.0 PL=0
MOVL C01078 V=800.0 PL=0
MOVL C01079 V=800.0 PL=0
MOVL C01080 V=800.0 PL=0
MOVL C01081 V=800.0 PL=0
MOVL C01082 V=800.0 PL=0
MOVL C01083 V=800.0 PL=0
MOVL C01084 V=800.0 PL=0
MOVL C01085 V=800.0 PL=0
MOVL C01086 V=800.0 PL=0
MOVL C01087 V=800.0 PL=0
MOVL C01088 V=800.0 PL=0
MOVL C01089 V=800.0 PL=0
MOVL C01090 V=800.0 PL=0
MOVL C01091 V=800.0 PL=0
MOVL C01092 V=800.0 PL=0
MOVL C01093 V=800.0 PL=0
MOVL C01094 V=800.0 PL=0
MOVL C01095 V=800.0 PL=0
MOVL C01096 V=800.0 PL=0
MOVL C01097 V=800.0 PL=0
MOVL C01098 V=800.0 PL=0
MOVL C01099 V=800.0 PL=0
MOVL C01100 V=800.0 PL=0
MOVL C01101 V=800.0 PL=0
MOVL C01102 V=800.0 PL=0
MOVL C01103 V=800.0 PL=0
MOVL C01104 V=800.0 PL=0
MOVL C01105 V=800.0 PL=0
MOVL C01106 V=800.0 PL=0
MOVL C01107 V=800.0 PL=0
MOVL C01108 V=800.0 PL=0
MOVL C01109 V=800.0 PL=0
MOVL C01110 V=800.0 PL=0
MOVL C01111 V=800.0 PL=0
MOVL C01112 V=800.0 PL=0
MOVL C01113 V=800.0 PL=0
MOVL C01114 V=800.0 PL=0
MOVL C01115 V=800.0 PL=0
MOVL C01116 V=800.0 PL=0
MOVL C01117 V=800.0 PL=0
MOVL C01118 V=800.0 PL=0
MOVL C01119 V=800.0 PL=0
MOVL C01120 V=800.0 PL=0
MOVL C01121 V=800.0 PL=0
MOVL C01122 V=800.0 PL=0
MOVL C01123 V=800.0 PL=0
MOVL C01124 V=800.0 PL=0
MOVL C01125 V=800.0 PL=0
MOVL C01126 V=800.0 PL=0
MOVL C01127 V=800.0 PL=0
MOVL C01128 V=800.0 PL=0
MOVL C01129 V=800.0 PL=0
MOVL C01130 V=800.0 PL=0
MOVL C01131 V=800.0 PL=0
MOVL C01132 V=800.0 PL=0
MOVL C01133 V=800.0 PL=0
MOVL C01134 V=800.0 PL=0
MOVL C01135 V=800.0 PL=0
MOVL C01136 V=800.0 PL=0
MOVL C01137 V=800.0 PL=0
MOVL C01138 V=800.0 PL=0
MOVL C01139 V=800.0 PL=0
MOVL C01140 V=800.0 PL=0
MOVL C01141 V=800.0 PL=0
MOVL C01142 V=800.0 PL=0
MOVL C01143 V=800.0 PL=0
MOVL C01144 V=800.0 PL=0
MOVL C01145 V=800.0 PL=0
MOVL C01146 V=800.0 PL=0
MOVL C01147 V=800.0 PL=0
MOVL C01148 V=800.0 PL=0
MOVL C01149 V=800.0 PL=0
MOVL C01150 V=800.0 PL=0
MOVL C01151 V=800.0 PL=0
MOVL C01152 V=800.0 PL=0
MOVL C01153 V=800.0 PL=0
MOVL C01154 V=800.0 PL=0
MOVL C01155 V=800.0 PL=0
MOVL C01156 V=800.0 PL=0
MOVL C01157 V=800.0 PL=0
MOVL C01158 V=800.0 PL=0
MOVL C01159 V=800.0 PL=0
MOVL C01160 V=800.0 PL=0
MOVL C01161 V=800.0 PL=0
MOVL C01162 V=800.0 PL=0
MOVL C01163 V=800.0 PL=0
MOVL C01164 V=800.0 PL=0
MOVL C01165 V=800.0 PL=0
MOVL C01166 V=800.0 PL=0
MOVL C01167 V=800.0 PL=0
MOVL C01168 V=800.0 PL=0
MOVL C01169 V=800.0 PL=0
MOVL C01170 V=800.0 PL=0
MOVL C01171 V=800.0 PL=0
MOVL C01172 V=800.0 PL=0
MOVL C01173 V=800.0 PL=0
MOVL C01174 V=800.0 PL=0
MOVL C01175 V=800.0 PL=0
MOVL C01176 V=800.0 PL=0
MOVL C01177 V=800.0 PL=0
MOVL C01178 V=800.0 PL=0
MOVL C01179 V=800.0 PL=0
MOVL C01180 V=800.0 PL=0
MOVL C01181 V=800.0 PL=0
MOVL C01182 V=800.0 PL=0
MOVL C01183 V=800.0 PL=0
MOVL C01184 V=800.0 PL=0
MOVL C01185 V=800.0 PL=0
MOVL C01186 V=800.0 PL=0
MOVL C01187 V=800.0 PL=0
MOVL C01188 V=800.0 PL=0
MOVL C01189 V=800.0 PL=0
MOVL C01190 V=800.0 PL=0
MOVL C01191 V=800.0 PL=0
MOVL C01192 V=800.0 PL=0
MOVL C01193 V=800.0 PL=0
MOVL C01194 V=800.0 PL=0
MOVL C01195 V=800.0 PL=0
MOVL C01196 V=800.0 PL=0
MOVL C01197 V=800.0 PL=0
MOVL C01198 V=800.0 PL=0
MOVL C01199 V=800.0 PL=0
MOVL C01200 V=800.0 PL=0
MOVL C01201 V=800.0 PL=0
MOVL C01202 V=800.0 PL=0
MOVL C01203 V=800.0 PL=0
MOVL C01204 V=800.0 PL=0
MOVL C01205 V=800.0 PL=0
MOVL C01206 V=800.0 PL=0
MOVL C01207 V=800.0 PL=0
MOVL C01208 V=800.0 PL=0
MOVL C01209 V=800.0 PL=0
MOVL C01210 V=800.0 PL=0
MOVL C01211 V=800.0 PL=0
MOVL C01212 V=800.0 PL=0
MOVL C01213 V=800.0 PL=0
MOVL C01214 V=800.0 PL=0
MOVL C01215 V=800.0 PL=0
MOVL C01216 V=800.0 PL=0
MOVL C01217 V=800.0 PL=0
MOVL C01218 V=800.0 PL=0
MOVL C01219 V=800.0 PL=0
MOVL C01220 V=800.0 PL=0
MOVL C01221 V=800.0 PL=0
MOVL C01222 V=800.0 PL=0
MOVL C01223 V=800.0 PL=0
MOVL C01224 V=800.0 PL=0
MOVL C01225 V=800.0 PL=0
MOVL C01226 V=800.0 PL=0
MOVL C01227 V=800.0 PL=0
MOVL C01228 V=800.0 PL=0
MOVL C01229 V=800.0 PL=0
MOVL C01230 V=800.0 PL=0
MOVL C01231 V=800.0 PL=0
MOVL C01232 V=800.0 PL=0
MOVL C01233 V=800.0 PL=0
MOVL C01234 V=800.0 PL=0
MOVL C01235 V=800.0 PL=0
MOVL C01236 V=800.0 PL=0
MOVL C01237 V=800.0 PL=0
MOVL C01238 V=800.0 PL=0
MOVL C01239 V=800.0 PL=0
MOVL C01240 V=800.0 PL=0
MOVL C01241 V=800.0 PL=0
MOVL C01242 V=800.0 PL=0
MOVL C01243 V=800.0 PL=0
MOVL C01244 V=800.0 PL=0
MOVL C01245 V=800.0 PL=0
MOVL C01246 V=800.0 PL=0
MOVL C01247 V=800.0 PL=0
MOVL C01248 V=800.0 PL=0
MOVL C01249 V=800.0 PL=0
MOVL C01250 V=800.0 PL=0
MOVL C01251 V=800.0 PL=0
MOVL C01252 V=800.0 PL=0
MOVL C01253 V=800.0 PL=0
MOVL C01254 V=800.0 PL=0
MOVL C01255 V=800.0 PL=0
MOVL C01256 V=800.0 PL=0
MOVL C01257 V=800.0 PL=0
MOVL C01258 V=800.0 PL=0
MOVL C01259 V=800.0 PL=0
MOVL C01260 V=800.0 PL=0
MOVL C01261 V=800.0 PL=0
MOVL C01262 V=800.0 PL=0
MOVL C01263 V=800.0 PL=0
MOVL C01264 V=800.0 PL=0
MOVL C01265 V=800.0 PL=0
MOVL C01266 V=800.0 PL=0
MOVL C01267 V=800.0 PL=0
MOVL C01268 V=800.0 PL=0
MOVL C01269 V=800.0 PL=0
MOVL C01270 V=800.0 PL=0
MOVL C01271 V=800.0 PL=0
MOVL C01272 V=800.0 PL=0
MOVL C01273 V=800.0 PL=0
MOVL C01274 V=800.0 PL=0
MOVL C01275 V=800.0 PL=0
MOVL C01276 V=800.0 PL=0
MOVL C01277 V=800.0 PL=0
MOVL C01278 V=800.0 PL=0
MOVL C01279 V=800.0 PL=0
MOVL C01280 V=800.0 PL=0
MOVL C01281 V=800.0 PL=0
MOVL C01282 V=800.0 PL=0
MOVL C01283 V=800.0 PL=0
MOVL C01284 V=800.0 PL=0
MOVL C01285 V=800.0 PL=0
MOVL C01286 V=800.0 PL=0
MOVL C01287 V=800.0 PL=0
MOVL C01288 V=800.0 PL=0
MOVL C01289 V=800.0 PL=0
MOVL C01290 V=800.0 PL=0
MOVL C01291 V=800.0 PL=0
MOVL C01292 V=800.0 PL=0
MOVL C01293 V=800.0 PL=0
MOVL C01294 V=800.0 PL=0
MOVL C01295 V=800.0 PL=0
MOVL C01296 V=800.0 PL=0
MOVL C01297 V=800.0 PL=0
MOVL C01298 V=800.0 PL=0
MOVL C01299 V=800.0 PL=0
MOVL C01300 V=800.0 PL=0
MOVL C01301 V=800.0 PL=0
MOVL C01302 V=800.0 PL=0
MOVL C01303 V=800.0 PL=0
MOVL C01304 V=800.0 PL=0
MOVL C01305 V=800.0 PL=0
MOVL C01306 V=800.0 PL=0
MOVL C01307 V=800.0 PL=0
MOVL C01308 V=800.0 PL=0
MOVL C01309 V=800.0 PL=0
MOVL C01310 V=800.0 PL=0
MOVL C01311 V=800.0 PL=0
MOVL C01312 V=800.0 PL=0
MOVL C01313 V=800.0 PL=0
MOVL C01314 V=800.0 PL=0
MOVL C01315 V=800.0 PL=0
MOVL C01316 V=800.0 PL=0
MOVL C01317 V=800.0 PL=0
MOVL C01318 V=800.0 PL=0
MOVL C01319 V=800.0 PL=0
MOVL C01320 V=800.0 PL=0
MOVL C01321 V=800.0 PL=0
MOVL C01322 V=800.0 PL=0
MOVL C01323 V=800.0 PL=0
MOVL C01324 V=800.0 PL=0
MOVL C01325 V=800.0 PL=0
MOVL C01326 V=800.0 PL=0
MOVL C01327 V=800.0 PL=0
MOVL C01328 V=800.0 PL=0
MOVL C01329 V=800.0 PL=0
MOVL C01330 V=800.0 PL=0
MOVL C01331 V=800.0 PL=0
MOVL C01332 V=800.0 PL=0
MOVL C01333 V=800.0 PL=0
MOVL C01334 V=800.0 PL=0
MOVL C01335 V=800.0 PL=0
MOVL C01336 V=800.0 PL=0
MOVL C01337 V=800.0 PL=0
MOVL C01338 V=800.0 PL=0
MOVL C01339 V=800.0 PL=0
MOVL C01340 V=800.0 PL=0
MOVL C01341 V=800.0 PL=0
MOVL C01342 V=800.0 PL=0
MOVL C01343 V=800.0 PL=0
MOVL C01344 V=800.0 PL=0
MOVL C01345 V=800.0 PL=0
MOVL C01346 V=800.0 PL=0
MOVL C01347 V=800.0 PL=0
MOVL C01348 V=800.0 PL=0
MOVL C01349 V=800.0 PL=0
MOVL C01350 V=800.0 PL=0
MOVL C01351 V=800.0 PL=0
MOVL C01352 V=800.0 PL=0
MOVL C01353 V=800.0 PL=0
MOVL C01354 V=800.0 PL=0
MOVL C01355 V=800.0 PL=0
MOVL C01356 V=800.0 PL=0
MOVL C01357 V=800.0 PL=0
MOVL C01358 V=800.0 PL=0
MOVL C01359 V=800.0 PL=0
MOVL C01360 V=800.0 PL=0
MOVL C01361 V=800.0 PL=0
MOVL C01362 V=800.0 PL=0
MOVL C01363 V=800.0 PL=0
MOVL C01364 V=800.0 PL=0
MOVL C01365 V=800.0 PL=0
MOVL C01366 V=800.0 PL=0
MOVL C01367 V=800.0 PL=0
MOVL C01368 V=800.0 PL=0
MOVL C01369 V=800.0 PL=0
MOVL C01370 V=800.0 PL=0
MOVL C01371 V=800.0 PL=0
MOVL C01372 V=800.0 PL=0
MOVL C01373 V=800.0 PL=0
MOVL C01374 V=800.0 PL=0
MOVL C01375 V=800.0 PL=0
MOVL C01376 V=800.0 PL=0
MOVL C01377 V=800.0 PL=0
MOVL C01378 V=800.0 PL=0
MOVL C01379 V=800.0 PL=0
MOVL C01380 V=800.0 PL=0
MOVL C01381 V=800.0 PL=0
MOVL C01382 V=800.0 PL=0
MOVL C01383 V=800.0 PL=0
MOVL C01384 V=800.0 PL=0
MOVL C01385 V=800.0 PL=0
MOVL C01386 V=800.0 PL=0
MOVL C01387 V=800.0 PL=0
MOVL C01388 V=800.0 PL=0
MOVL C01389 V=800.0 PL=0
MOVL C01390 V=800.0 PL=0
MOVL C01391 V=800.0 PL=0
MOVL C01392 V=800.0 PL=0
MOVL C01393 V=800.0 PL=0
MOVL C01394 V=800.0 PL=0
MOVL C01395 V=800.0 PL=0
MOVL C01396 V=800.0 PL=0
MOVL C01397 V=800.0 PL=0
MOVL C01398 V=800.0 PL=0
MOVL C01399 V=800.0 PL=0
MOVL C01400 V=800.0 PL=0
MOVL C01401 V=800.0 PL=0
MOVL C01402 V=800.0 PL=0
MOVL C01403 V=800.0 PL=0
MOVL C01404 V=800.0 PL=0
MOVL C01405 V=800.0 PL=0
MOVL C01406 V=800.0 PL=0
MOVL C01407 V=800.0 PL=0
MOVL C01408 V=800.0 PL=0
MOVL C01409 V=800.0 PL=0
MOVL C01410 V=800.0 PL=0
MOVL C01411 V=800.0 PL=0
MOVL C01412 V=800.0 PL=0
MOVL C01413 V=800.0 PL=0
MOVL C01414 V=800.0 PL=0
MOVL C01415 V=800.0 PL=0
MOVL C01416 V=800.0 PL=0
MOVL C01417 V=800.0 PL=0
MOVL C01418 V=800.0 PL=0
MOVL C01419 V=800.0 PL=0
MOVL C01420 V=800.0 PL=0
MOVL C01421 V=800.0 PL=0
MOVL C01422 V=800.0 PL=0
MOVL C01423 V=800.0 PL=0
MOVL C01424 V=800.0 PL=0
MOVL C01425 V=800.0 PL=0
MOVL C01426 V=800.0 PL=0
MOVL C01427 V=800.0 PL=0
MOVL C01428 V=800.0 PL=0
MOVL C01429 V=800.0 PL=0
MOVL C01430 V=800.0 PL=0
MOVL C01431 V=800.0 PL=0
MOVL C01432 V=800.0 PL=0
MOVL C01433 V=800.0 PL=0
MOVL C01434 V=800.0 PL=0
MOVL C01435 V=800.0 PL=0
MOVL C01436 V=800.0 PL=0
MOVL C01437 V=800.0 PL=0
MOVL C01438 V=800.0 PL=0
MOVL C01439 V=800.0 PL=0
MOVL C01440 V=800.0 PL=0
MOVL C01441 V=800.0 PL=0
MOVL C01442 V=800.0 PL=0
MOVL C01443 V=800.0 PL=0
MOVL C01444 V=800.0 PL=0
MOVL C01445 V=800.0 PL=0
MOVL C01446 V=800.0 PL=0
MOVL C01447 V=800.0 PL=0
MOVL C01448 V=800.0 PL=0
MOVL C01449 V=800.0 PL=0
MOVL C01450 V=800.0 PL=0
MOVL C01451 V=800.0 PL=0
MOVL C01452 V=800.0 PL=0
MOVL C01453 V=800.0 PL=0
MOVL C01454 V=800.0 PL=0
MOVL C01455 V=800.0 PL=0
MOVL C01456 V=800.0 PL=0
MOVL C01457 V=800.0 PL=0
MOVL C01458 V=800.0 PL=0
MOVL C01459 V=800.0 PL=0
MOVL C01460 V=800.0 PL=0
MOVL C01461 V=800.0 PL=0
MOVL C01462 V=800.0 PL=0
MOVL C01463 V=800.0 PL=0
MOVL C01464 V=800.0 PL=0
MOVL C01465 V=800.0 PL=0
MOVL C01466 V=800.0 PL=0
MOVL C01467 V=800.0 PL=0
MOVL C01468 V=800.0 PL=0
MOVL C01469 V=800.0 PL=0
MOVL C01470 V=800.0 PL=0
MOVL C01471 V=800.0 PL=0
MOVL C01472 V=800.0 PL=0
MOVL C01473 V=800.0 PL=0
MOVL C01474 V=800.0 PL=0
MOVL C01475 V=800.0 PL=0
MOVL C01476 V=800.0 PL=0
MOVL C01477 V=800.0 PL=0
MOVL C01478 V=800.0 PL=0
MOVL C01479 V=800.0 PL=0
MOVL C01480 V=800.0 PL=0
MOVL C01481 V=800.0 PL=0
MOVL C01482 V=800.0 PL=0
MOVL C01483 V=800.0 PL=0
MOVL C01484 V=800.0 PL=0
MOVL C01485 V=800.0 PL=0
MOVL C01486 V=800.0 PL=0
MOVL C01487 V=800.0 PL=0
MOVL C01488 V=800.0 PL=0
MOVL C01489 V=800.0 PL=0
MOVL C01490 V=800.0 PL=0
MOVL C01491 V=800.0 PL=0
MOVL C01492 V=800.0 PL=0
MOVL C01493 V=800.0 PL=0
MOVL C01494 V=800.0 PL=0
MOVL C01495 V=800.0 PL=0
MOVL C01496 V=800.0 PL=0
MOVL C01497 V=800.0 PL=0
MOVL C01498 V=800.0 PL=0
MOVL C01499 V=800.0 PL=0
MOVL C01500 V=800.0 PL=0
MOVL C01501 V=800.0 PL=0
MOVL C01502 V=800.0 PL=0
MOVL C01503 V=800.0 PL=0
MOVL C01504 V=800.0 PL=0
MOVL C01505 V=800.0 PL=0
MOVL C01506 V=800.0 PL=0
MOVL C01507 V=800.0 PL=0
MOVL C01508 V=800.0 PL=0
MOVL C01509 V=800.0 PL=0
MOVL C01510 V=800.0 PL=0
MOVL C01511 V=800.0 PL=0
MOVL C01512 V=800.0 PL=0
MOVL C01513 V=800.0 PL=0
MOVL C01514 V=800.0 PL=0
MOVL C01515 V=800.0 PL=0
MOVL C01516 V=800.0 PL=0
MOVL C01517 V=800.0 PL=0
MOVL C01518 V=800.0 PL=0
MOVL C01519 V=800.0 PL=0
MOVL C01520 V=800.0 PL=0
MOVL C01521 V=800.0 PL=0
MOVL C01522 V=800.0 PL=0
MOVL C01523 V=800.0 PL=0
MOVL C01524 V=800.0 PL=0
MOVL C01525 V=800.0 PL=0
MOVL C01526 V=800.0 PL=0
MOVL C01527 V=800.0 PL=0
MOVL C01528 V=800.0 PL=0
MOVL C01529 V=800.0 PL=0
MOVL C01530 V=800.0 PL=0
MOVL C01531 V=800.0 PL=0
MOVL C01532 V=800.0 PL=0
MOVL C01533 V=800.0 PL=0
MOVL C01534 V=800.0 PL=0
MOVL C01535 V=800.0 PL=0
MOVL C01536 V=800.0 PL=0
MOVL C01537 V=800.0 PL=0
MOVL C01538 V=800.0 PL=0
MOVL C01539 V=800.0 PL=0
MOVL C01540 V=800.0 PL=0
MOVL C01541 V=800.0 PL=0
MOVL C01542 V=800.0 PL=0
MOVL C01543 V=800.0 PL=0
MOVL C01544 V=800.0 PL=0
MOVL C01545 V=800.0 PL=0
MOVL C01546 V=800.0 PL=0
MOVL C01547 V=800.0 PL=0
MOVL C01548 V=800.0 PL=0
MOVL C01549 V=800.0 PL=0
MOVL C01550 V=800.0 PL=0
MOVL C01551 V=800.0 PL=0
MOVL C01552 V=800.0 PL=0
MOVL C01553 V=800.0 PL=0
MOVL C01554 V=800.0 PL=0
MOVL C01555 V=800.0 PL=0
MOVL C01556 V=800.0 PL=0
MOVL C01557 V=800.0 PL=0
MOVL C01558 V=800.0 PL=0
MOVL C01559 V=800.0 PL=0
MOVL C01560 V=800.0 PL=0
MOVL C01561 V=800.0 PL=0
MOVL C01562 V=800.0 PL=0
MOVL C01563 V=800.0 PL=0
MOVL C01564 V=800.0 PL=0
MOVL C01565 V=800.0 PL=0
MOVL C01566 V=800.0 PL=0
MOVL C01567 V=800.0 PL=0
MOVL C01568 V=800.0 PL=0
MOVL C01569 V=800.0 PL=0
MOVL C01570 V=800.0 PL=0
MOVL C01571 V=800.0 PL=0
MOVL C01572 V=800.0 PL=0
MOVL C01573 V=800.0 PL=0
MOVL C01574 V=800.0 PL=0
MOVL C01575 V=800.0 PL=0
MOVL C01576 V=800.0 PL=0
MOVL C01577 V=800.0 PL=0
MOVL C01578 V=800.0 PL=0
MOVL C01579 V=800.0 PL=0
MOVL C01580 V=800.0 PL=0
MOVL C01581 V=800.0 PL=0
MOVL C01582 V=800.0 PL=0
MOVL C01583 V=800.0 PL=0
MOVL C01584 V=800.0 PL=0
MOVL C01585 V=800.0 PL=0
MOVL C01586 V=800.0 PL=0
MOVL C01587 V=800.0 PL=0
MOVL C01588 V=800.0 PL=0
MOVL C01589 V=800.0 PL=0
MOVL C01590 V=800.0 PL=0
MOVL C01591 V=800.0 PL=0
MOVL C01592 V=800.0 PL=0
MOVL C01593 V=800.0 PL=0
MOVL C01594 V=800.0 PL=0
MOVL C01595 V=800.0 PL=0
MOVL C01596 V=800.0 PL=0
MOVL C01597 V=800.0 PL=0
MOVL C01598 V=800.0 PL=0
MOVL C01599 V=800.0 PL=0
MOVL C01600 V=800.0 PL=0
MOVL C01601 V=800.0 PL=0
MOVL C01602 V=800.0 PL=0
MOVL C01603 V=800.0 PL=0
MOVL C01604 V=800.0 PL=0
MOVL C01605 V=800.0 PL=0
MOVL C01606 V=800.0 PL=0
MOVL C01607 V=800.0 PL=0
MOVL C01608 V=800.0 PL=0
MOVL C01609 V=800.0 PL=0
MOVL C01610 V=800.0 PL=0
MOVL C01611 V=800.0 PL=0
MOVL C01612 V=800.0 PL=0
MOVL C01613 V=800.0 PL=0
MOVL C01614 V=800.0 PL=0
MOVL C01615 V=800.0 PL=0
MOVL C01616 V=800.0 PL=0
MOVL C01617 V=800.0 PL=0
MOVL C01618 V=800.0 PL=0
MOVL C01619 V=800.0 PL=0
MOVL C01620 V=800.0 PL=0
MOVL C01621 V=800.0 PL=0
MOVL C01622 V=800.0 PL=0
MOVL C01623 V=800.0 PL=0
MOVL C01624 V=800.0 PL=0
MOVL C01625 V=800.0 PL=0
MOVL C01626 V=800.0 PL=0
MOVL C01627 V=800.0 PL=0
MOVL C01628 V=800.0 PL=0
MOVL C01629 V=800.0 PL=0
MOVL C01630 V=800.0 PL=0
MOVL C01631 V=800.0 PL=0
MOVL C01632 V=800.0 PL=0
MOVL C01633 V=800.0 PL=0
MOVL C01634 V=800.0 PL=0
MOVL C01635 V=800.0 PL=0
MOVL C01636 V=800.0 PL=0
MOVL C01637 V=800.0 PL=0
MOVL C01638 V=800.0 PL=0
MOVL C01639 V=800.0 PL=0
MOVL C01640 V=800.0 PL=0
MOVL C01641 V=800.0 PL=0
MOVL C01642 V=800.0 PL=0
MOVL C01643 V=800.0 PL=0
MOVL C01644 V=800.0 PL=0
MOVL C01645 V=800.0 PL=0
MOVL C01646 V=800.0 PL=0
MOVL C01647 V=800.0 PL=0
MOVL C01648 V=800.0 PL=0
MOVL C01649 V=800.0 PL=0
MOVL C01650 V=800.0 PL=0
MOVL C01651 V=800.0 PL=0
MOVL C01652 V=800.0 PL=0
MOVL C01653 V=800.0 PL=0
MOVL C01654 V=800.0 PL=0
MOVL C01655 V=800.0 PL=0
MOVL C01656 V=800.0 PL=0
MOVL C01657 V=800.0 PL=0
MOVL C01658 V=800.0 PL=0
MOVL C01659 V=800.0 PL=0
MOVL C01660 V=800.0 PL=0
MOVL C01661 V=800.0 PL=0
MOVL C01662 V=800.0 PL=0
MOVL C01663 V=800.0 PL=0
MOVL C01664 V=800.0 PL=0
MOVL C01665 V=800.0 PL=0
MOVL C01666 V=800.0 PL=0
MOVL C01667 V=800.0 PL=0
MOVL C01668 V=800.0 PL=0
MOVL C01669 V=800.0 PL=0
MOVL C01670 V=800.0 PL=0
MOVL C01671 V=800.0 PL=0
MOVL C01672 V=800.0 PL=0
MOVL C01673 V=800.0 PL=0
MOVL C01674 V=800.0 PL=0
MOVL C01675 V=800.0 PL=0
MOVL C01676 V=800.0 PL=0
MOVL C01677 V=800.0 PL=0
MOVL C01678 V=800.0 PL=0
MOVL C01679 V=800.0 PL=0
MOVL C01680 V=800.0 PL=0
MOVL C01681 V=800.0 PL=0
MOVL C01682 V=800.0 PL=0
MOVL C01683 V=800.0 PL=0
MOVL C01684 V=800.0 PL=0
MOVL C01685 V=800.0 PL=0
MOVL C01686 V=800.0 PL=0
MOVL C01687 V=800.0 PL=0
MOVL C01688 V=800.0 PL=0
MOVL C01689 V=800.0 PL=0
MOVL C01690 V=800.0 PL=0
MOVL C01691 V=800.0 PL=0
MOVL C01692 V=800.0 PL=0
MOVL C01693 V=800.0 PL=0
MOVL C01694 V=800.0 PL=0
MOVL C01695 V=800.0 PL=0
MOVL C01696 V=800.0 PL=0
MOVL C01697 V=800.0 PL=0
MOVL C01698 V=800.0 PL=0
MOVL C01699 V=800.0 PL=0
MOVL C01700 V=800.0 PL=0
MOVL C01701 V=800.0 PL=0
MOVL C01702 V=800.0 PL=0
MOVL C01703 V=800.0 PL=0
MOVL C01704 V=800.0 PL=0
MOVL C01705 V=800.0 PL=0
MOVL C01706 V=800.0 PL=0
MOVL C01707 V=800.0 PL=0
MOVL C01708 V=800.0 PL=0
MOVL C01709 V=800.0 PL=0
MOVL C01710 V=800.0 PL=0
MOVL C01711 V=800.0 PL=0
MOVL C01712 V=800.0 PL=0
MOVL C01713 V=800.0 PL=0
MOVL C01714 V=800.0 PL=0
MOVL C01715 V=800.0 PL=0
MOVL C01716 V=800.0 PL=0
MOVL C01717 V=800.0 PL=0
MOVL C01718 V=800.0 PL=0
MOVL C01719 V=800.0 PL=0
MOVL C01720 V=800.0 PL=0
MOVL C01721 V=800.0 PL=0
MOVL C01722 V=800.0 PL=0
MOVL C01723 V=800.0 PL=0
MOVL C01724 V=800.0 PL=0
MOVL C01725 V=800.0 PL=0
MOVL C01726 V=800.0 PL=0
MOVL C01727 V=800.0 PL=0
MOVL C01728 V=800.0 PL=0
MOVL C01729 V=800.0 PL=0
MOVL C01730 V=800.0 PL=0
MOVL C01731 V=800.0 PL=0
MOVL C01732 V=800.0 PL=0
MOVL C01733 V=800.0 PL=0
MOVL C01734 V=800.0 PL=0
MOVL C01735 V=800.0 PL=0
MOVL C01736 V=800.0 PL=0
MOVL C01737 V=800.0 PL=0
MOVL C01738 V=800.0 PL=0
MOVL C01739 V=800.0 PL=0
MOVL C01740 V=800.0 PL=0
MOVL C01741 V=800.0 PL=0
MOVL C01742 V=800.0 PL=0
MOVL C01743 V=800.0 PL=0
MOVL C01744 V=800.0 PL=0
MOVL C01745 V=800.0 PL=0
MOVL C01746 V=800.0 PL=0
MOVL C01747 V=800.0 PL=0
MOVL C01748 V=800.0 PL=0
MOVL C01749 V=800.0 PL=0
MOVL C01750 V=800.0 PL=0
MOVL C01751 V=800.0 PL=0
MOVL C01752 V=800.0 PL=0
MOVL C01753 V=800.0 PL=0
MOVL C01754 V=800.0 PL=0
MOVL C01755 V=800.0 PL=0
MOVL C01756 V=800.0 PL=0
MOVL C01757 V=800.0 PL=0
MOVL C01758 V=800.0 PL=0
MOVL C01759 V=800.0 PL=0
MOVL C01760 V=800.0 PL=0
MOVL C01761 V=800.0 PL=0
MOVL C01762 V=800.0 PL=0
MOVL C01763 V=800.0 PL=0
MOVL C01764 V=800.0 PL=0
MOVL C01765 V=800.0 PL=0
MOVL C01766 V=800.0 PL=0
MOVL C01767 V=800.0 PL=0
MOVL C01768 V=800.0 PL=0
MOVL C01769 V=800.0 PL=0
MOVL C01770 V=800.0 PL=0
MOVL C01771 V=800.0 PL=0
MOVL C01772 V=800.0 PL=0
MOVL C01773 V=800.0 PL=0
MOVL C01774 V=800.0 PL=0
MOVL C01775 V=800.0 PL=0
MOVL C01776 V=800.0 PL=0
MOVL C01777 V=800.0 PL=0
MOVL C01778 V=800.0 PL=0
MOVL C01779 V=800.0 PL=0
MOVL C01780 V=800.0 PL=0
MOVL C01781 V=800.0 PL=0
MOVL C01782 V=800.0 PL=0
MOVL C01783 V=800.0 PL=0
MOVL C01784 V=800.0 PL=0
MOVL C01785 V=800.0 PL=0
MOVL C01786 V=800.0 PL=0
MOVL C01787 V=800.0 PL=0
MOVL C01788 V=800.0 PL=0
MOVL C01789 V=800.0 PL=0
MOVL C01790 V=800.0 PL=0
MOVL C01791 V=800.0 PL=0
MOVL C01792 V=800.0 PL=0
MOVL C01793 V=800.0 PL=0
MOVL C01794 V=800.0 PL=0
MOVL C01795 V=800.0 PL=0
MOVL C01796 V=800.0 PL=0
MOVL C01797 V=800.0 PL=0
MOVL C01798 V=800.0 PL=0
MOVL C01799 V=800.0 PL=0
MOVL C01800 V=800.0 PL=0
MOVL C01801 V=800.0 PL=0
MOVL C01802 V=800.0 PL=0
MOVL C01803 V=800.0 PL=0
MOVL C01804 V=800.0 PL=0
MOVL C01805 V=800.0 PL=0
MOVL C01806 V=800.0 PL=0
MOVL C01807 V=800.0 PL=0
MOVL C01808 V=800.0 PL=0
MOVL C01809 V=800.0 PL=0
MOVL C01810 V=800.0 PL=0
MOVL C01811 V=800.0 PL=0
MOVL C01812 V=800.0 PL=0
MOVL C01813 V=800.0 PL=0
MOVL C01814 V=800.0 PL=0
MOVL C01815 V=800.0 PL=0
MOVL C01816 V=800.0 PL=0
MOVL C01817 V=800.0 PL=0
MOVL C01818 V=800.0 PL=0
MOVL C01819 V=800.0 PL=0
MOVL C01820 V=800.0 PL=0
MOVL C01821 V=800.0 PL=0
MOVL C01822 V=800.0 PL=0
MOVL C01823 V=800.0 PL=0
MOVL C01824 V=800.0 PL=0
MOVL C01825 V=800.0 PL=0
MOVL C01826 V=800.0 PL=0
MOVL C01827 V=800.0 PL=0
MOVL C01828 V=800.0 PL=0
MOVL C01829 V=800.0 PL=0
MOVL C01830 V=800.0 PL=0
MOVL C01831 V=800.0 PL=0
MOVL C01832 V=800.0 PL=0
MOVL C01833 V=800.0 PL=0
MOVL C01834 V=800.0 PL=0
MOVL C01835 V=800.0 PL=0
MOVL C01836 V=800.0 PL=0
MOVL C01837 V=800.0 PL=0
MOVL C01838 V=800.0 PL=0
MOVL C01839 V=800.0 PL=0
MOVL C01840 V=800.0 PL=0
MOVL C01841 V=800.0 PL=0
MOVL C01842 V=800.0 PL=0
MOVL C01843 V=800.0 PL=0
MOVL C01844 V=800.0 PL=0
MOVL C01845 V=800.0 PL=0
MOVL C01846 V=800.0 PL=0
MOVL C01847 V=800.0 PL=0
MOVL C01848 V=800.0 PL=0
MOVL C01849 V=800.0 PL=0
MOVL C01850 V=800.0 PL=0
MOVL C01851 V=800.0 PL=0
MOVL C01852 V=800.0 PL=0
MOVL C01853 V=800.0 PL=0
MOVL C01854 V=800.0 PL=0
MOVL C01855 V=800.0 PL=0
MOVL C01856 V=800.0 PL=0
MOVL C01857 V=800.0 PL=0
MOVL C01858 V=800.0 PL=0
MOVL C01859 V=800.0 PL=0
MOVL C01860 V=800.0 PL=0
MOVL C01861 V=800.0 PL=0
MOVL C01862 V=800.0 PL=0
MOVL C01863 V=800.0 PL=0
MOVL C01864 V=800.0 PL=0
MOVL C01865 V=800.0 PL=0
MOVL C01866 V=800.0 PL=0
MOVL C01867 V=800.0 PL=0
MOVL C01868 V=800.0 PL=0
MOVL C01869 V=800.0 PL=0
MOVL C01870 V=800.0 PL=0
MOVL C01871 V=800.0 PL=0
MOVL C01872 V=800.0 PL=0
MOVL C01873 V=800.0 PL=0
MOVL C01874 V=800.0 PL=0
MOVL C01875 V=800.0 PL=0
MOVL C01876 V=800.0 PL=0
MOVL C01877 V=800.0 PL=0
MOVL C01878 V=800.0 PL=0
MOVL C01879 V=800.0 PL=0
MOVL C01880 V=800.0 PL=0
MOVL C01881 V=800.0 PL=0
MOVL C01882 V=800.0 PL=0
MOVL C01883 V=800.0 PL=0
MOVL C01884 V=800.0 PL=0
MOVL C01885 V=800.0 PL=0
MOVL C01886 V=800.0 PL=0
MOVL C01887 V=800.0 PL=0
MOVL C01888 V=800.0 PL=0
MOVL C01889 V=800.0 PL=0
MOVL C01890 V=800.0 PL=0
MOVL C01891 V=800.0 PL=0
MOVL C01892 V=800.0 PL=0
MOVL C01893 V=800.0 PL=0
MOVL C01894 V=800.0 PL=0
MOVL C01895 V=800.0 PL=0
MOVL C01896 V=800.0 PL=0
MOVL C01897 V=800.0 PL=0
MOVL C01898 V=800.0 PL=0
MOVL C01899 V=800.0 PL=0
MOVL C01900 V=800.0 PL=0
MOVL C01901 V=800.0 PL=0
MOVL C01902 V=800.0 PL=0
MOVL C01903 V=800.0 PL=0
MOVL C01904 V=800.0 PL=0
MOVL C01905 V=800.0 PL=0
MOVL C01906 V=800.0 PL=0
MOVL C01907 V=800.0 PL=0
MOVL C01908 V=800.0 PL=0
MOVL C01909 V=800.0 PL=0
MOVL C01910 V=800.0 PL=0
MOVL C01911 V=800.0 PL=0
MOVL C01912 V=800.0 PL=0
MOVL C01913 V=800.0 PL=0
MOVL C01914 V=800.0 PL=0
MOVL C01915 V=800.0 PL=0
MOVL C01916 V=800.0 PL=0
MOVL C01917 V=800.0 PL=0
MOVL C01918 V=800.0 PL=0
MOVL C01919 V=800.0 PL=0
MOVL C01920 V=800.0 PL=0
MOVL C01921 V=800.0 PL=0
MOVL C01922 V=800.0 PL=0
MOVL C01923 V=800.0 PL=0
MOVL C01924 V=800.0 PL=0
MOVL C01925 V=800.0 PL=0
MOVL C01926 V=800.0 PL=0
MOVL C01927 V=800.0 PL=0
MOVL C01928 V=800.0 PL=0
MOVL C01929 V=800.0 PL=0
MOVL C01930 V=800.0 PL=0
MOVL C01931 V=800.0 PL=0
MOVL C01932 V=800.0 PL=0
MOVL C01933 V=800.0 PL=0
MOVL C01934 V=800.0 PL=0
MOVL C01935 V=800.0 PL=0
MOVL C01936 V=800.0 PL=0
MOVL C01937 V=800.0 PL=0
MOVL C01938 V=800.0 PL=0
MOVL C01939 V=800.0 PL=0
MOVL C01940 V=800.0 PL=0
MOVL C01941 V=800.0 PL=0
MOVL C01942 V=800.0 PL=0
MOVL C01943 V=800.0 PL=0
MOVL C01944 V=800.0 PL=0
MOVL C01945 V=800.0 PL=0
MOVL C01946 V=800.0 PL=0
MOVL C01947 V=800.0 PL=0
MOVL C01948 V=800.0 PL=0
MOVL C01949 V=800.0 PL=0
MOVL C01950 V=800.0 PL=0
MOVL C01951 V=800.0 PL=0
MOVL C01952 V=800.0 PL=0
MOVL C01953 V=800.0 PL=0
MOVL C01954 V=800.0 PL=0
MOVL C01955 V=800.0 PL=0
MOVL C01956 V=800.0 PL=0
MOVL C01957 V=800.0 PL=0
MOVL C01958 V=800.0 PL=0
MOVL C01959 V=800.0 PL=0
MOVL C01960 V=800.0 PL=0
MOVL C01961 V=800.0 PL=0
MOVL C01962 V=800.0 PL=0
MOVL C01963 V=800.0 PL=0
MOVL C01964 V=800.0 PL=0
MOVL C01965 V=800.0 PL=0
MOVL C01966 V=800.0 PL=0
MOVL C01967 V=800.0 PL=0
MOVL C01968 V=800.0 PL=0
MOVL C01969 V=800.0 PL=0
MOVL C01970 V=800.0 PL=0
MOVL C01971 V=800.0 PL=0
MOVL C01972 V=800.0 PL=0
MOVL C01973 V=800.0 PL=0
MOVL C01974 V=800.0 PL=0
MOVL C01975 V=800.0 PL=0
MOVL C01976 V=800.0 PL=0
MOVL C01977 V=800.0 PL=0
MOVL C01978 V=800.0 PL=0
MOVL C01979 V=800.0 PL=0
MOVL C01980 V=800.0 PL=0
MOVL C01981 V=800.0 PL=0
MOVL C01982 V=800.0 PL=0
MOVL C01983 V=800.0 PL=0
MOVL C01984 V=800.0 PL=0
MOVL C01985 V=800.0 PL=0
MOVL C01986 V=800.0 PL=0
MOVL C01987 V=800.0 PL=0
MOVL C01988 V=800.0 PL=0
MOVL C01989 V=800.0 PL=0
MOVL C01990 V=800.0 PL=0
MOVL C01991 V=800.0 PL=0
MOVL C01992 V=800.0 PL=0
MOVL C01993 V=800.0 PL=0
MOVL C01994 V=800.0 PL=0
MOVL C01995 V=800.0 PL=0
MOVL C01996 V=800.0 PL=0
MOVL C01997 V=800.0 PL=0
MOVL C01998 V=800.0 PL=0
MOVL C01999 V=800.0 PL=0
MOVL C02000 V=800.0 PL=0
MOVL C02001 V=800.0 PL=0
MOVL C02002 V=800.0 PL=0
MOVL C02003 V=800.0 PL=0
MOVL C02004 V=800.0 PL=0
MOVL C02005 V=800.0 PL=0
MOVL C02006 V=800.0 PL=0
MOVL C02007 V=800.0 PL=0
MOVL C02008 V=800.0 PL=0
MOVL C02009 V=800.0 PL=0
MOVL C02010 V=800.0 PL=0
MOVL C02011 V=800.0 PL=0
MOVL C02012 V=800.0 PL=0
MOVL C02013 V=800.0 PL=0
